Yaskawa INFORM job: A_ROOF_SIDE_0617_2_PAINT_38.JBI

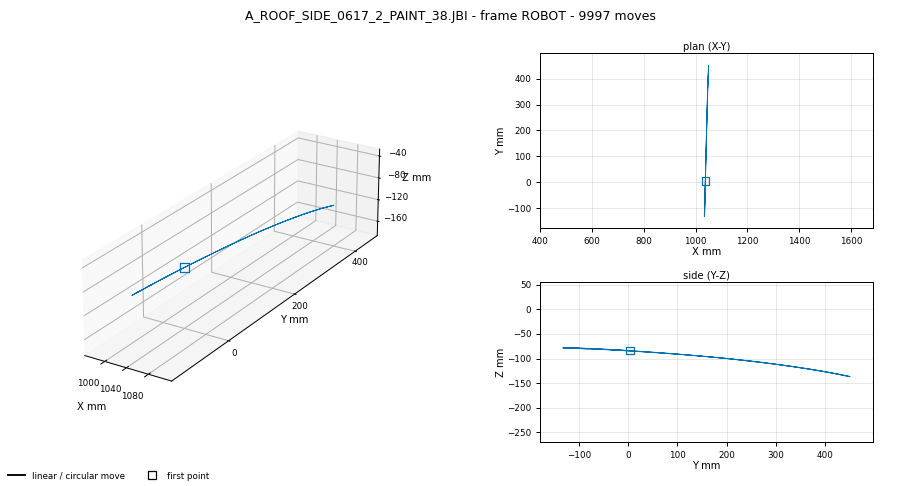
[picture p0: tool path of A_ROOF_SIDE_0617_2_PAINT_38.JBI in frame ROBOT, 9997 of 9997 moves have a stored position in this frame; points joined in program order, loops and branches not executed]
/JOB
//NAME A_ROOF_SIDE_0617_2_PAINT38
//POS
///NPOS 9997,0,0,0,0,0
///TOOL 1
///USER 0
///POSTYPE ROBOT
///RECTAN
///RCONF 1,0,0,0,0,0,0,0,0,0,0,0,0,0,0,0,0,0,0,0,0,0,0,0
C00000=1038.602,4.490,-83.697,169.159,38.320,157.198
C00001=1038.595,4.241,-83.682,169.157,38.319,157.198
C00002=1038.590,3.992,-83.668,169.155,38.320,157.198
C00003=1038.583,3.742,-83.653,169.153,38.319,157.198
C00004=1038.577,3.493,-83.638,169.151,38.318,157.198
C00005=1038.570,3.243,-83.622,169.149,38.318,157.198
C00006=1038.564,2.994,-83.607,169.147,38.318,157.198
C00007=1038.557,2.744,-83.592,169.145,38.317,157.197
C00008=1038.552,2.495,-83.578,169.142,38.317,157.197
C00009=1038.545,2.246,-83.563,169.140,38.317,157.197
C00010=1038.539,1.996,-83.548,169.138,38.316,157.197
C00011=1038.532,1.746,-83.533,169.136,38.316,157.197
C00012=1038.526,1.497,-83.518,169.134,38.315,157.197
C00013=1038.519,1.248,-83.502,169.132,38.315,157.197
C00014=1038.514,0.999,-83.487,169.130,38.315,157.197
C00015=1038.507,0.749,-83.473,169.128,38.314,157.197
C00016=1038.501,0.499,-83.458,169.125,38.314,157.196
C00017=1038.495,0.249,-83.442,169.123,38.314,157.196
C00018=1038.489,-0.000,-83.427,169.121,38.313,157.196
C00019=1038.483,-0.249,-83.413,169.119,38.313,157.196
C00020=1038.477,-0.499,-83.398,169.116,38.313,157.196
C00021=1038.470,-0.749,-83.383,169.114,38.312,157.196
C00022=1038.464,-0.998,-83.368,169.112,38.312,157.196
C00023=1038.458,-1.247,-83.353,169.110,38.311,157.196
C00024=1038.452,-1.497,-83.338,169.108,38.311,157.196
C00025=1038.445,-1.747,-83.323,169.106,38.311,157.196
C00026=1038.439,-1.996,-83.308,169.104,38.310,157.195
C00027=1038.433,-2.245,-83.294,169.102,38.310,157.195
C00028=1038.427,-2.495,-83.279,169.100,38.310,157.195
C00029=1038.420,-2.744,-83.264,169.098,38.309,157.195
C00030=1038.414,-2.994,-83.249,169.096,38.309,157.195
C00031=1038.407,-3.278,-83.233,169.092,38.308,157.195
C00032=1038.400,-3.560,-83.215,169.090,38.308,157.195
C00033=1038.393,-3.844,-83.198,169.087,38.308,157.195
C00034=1038.385,-4.127,-83.183,169.085,38.307,157.194
C00035=1038.379,-4.377,-83.168,169.083,38.307,157.194
C00036=1038.373,-4.627,-83.153,169.081,38.307,157.194
C00037=1038.366,-4.876,-83.138,169.079,38.307,157.194
C00038=1038.360,-5.125,-83.124,169.076,38.306,157.194
C00039=1038.354,-5.375,-83.110,169.074,38.306,157.194
C00040=1038.347,-5.625,-83.095,169.072,38.306,157.194
C00041=1038.340,-5.874,-83.080,169.070,38.306,157.194
C00042=1038.334,-6.123,-83.066,169.068,38.305,157.194
C00043=1038.328,-6.373,-83.051,169.066,38.306,157.194
C00044=1038.321,-6.623,-83.037,169.064,38.305,157.194
C00045=1038.315,-6.873,-83.022,169.061,38.304,157.193
C00046=1038.309,-7.122,-83.008,169.058,38.305,157.193
C00047=1038.303,-7.371,-82.993,169.056,38.304,157.193
C00048=1038.296,-7.621,-82.979,169.054,38.304,157.193
C00049=1038.290,-7.870,-82.965,169.052,38.304,157.193
C00050=1038.284,-8.120,-82.950,169.050,38.304,157.193
C00051=1038.277,-8.369,-82.935,169.048,38.303,157.193
C00052=1038.271,-8.619,-82.921,169.046,38.303,157.193
C00053=1038.265,-8.868,-82.906,169.043,38.303,157.193
C00054=1038.258,-9.118,-82.892,169.041,38.303,157.193
C00055=1038.252,-9.367,-82.877,169.039,38.302,157.193
C00056=1038.246,-9.617,-82.863,169.037,38.302,157.192
C00057=1038.239,-9.866,-82.849,169.035,38.302,157.192
C00058=1038.233,-10.115,-82.834,169.033,38.301,157.192
C00059=1038.227,-10.365,-82.820,169.030,38.301,157.192
C00060=1038.220,-10.615,-82.806,169.027,38.301,157.192
C00061=1038.214,-10.864,-82.791,169.025,38.301,157.192
C00062=1038.208,-11.114,-82.777,169.023,38.300,157.192
C00063=1038.201,-11.363,-82.763,169.021,38.300,157.192
C00064=1038.195,-11.613,-82.749,169.019,38.300,157.192
C00065=1038.189,-11.863,-82.734,169.017,38.299,157.192
C00066=1038.182,-12.111,-82.720,169.015,38.299,157.192
C00067=1038.176,-12.362,-82.706,169.012,38.299,157.191
C00068=1038.170,-12.611,-82.691,169.010,38.299,157.191
C00069=1038.163,-12.860,-82.677,169.008,38.298,157.191
C00070=1038.157,-13.110,-82.662,169.006,38.299,157.191
C00071=1038.151,-13.359,-82.648,169.004,38.298,157.191
C00072=1038.145,-13.609,-82.634,169.002,38.298,157.191
C00073=1038.139,-13.858,-82.620,168.998,38.298,157.191
C00074=1038.132,-14.108,-82.606,168.996,38.298,157.191
C00075=1038.126,-14.358,-82.591,168.994,38.297,157.191
C00076=1038.120,-14.607,-82.577,168.992,38.297,157.191
C00077=1038.113,-14.857,-82.563,168.990,38.297,157.191
C00078=1038.107,-15.105,-82.548,168.988,38.296,157.190
C00079=1038.101,-15.356,-82.534,168.985,38.296,157.190
C00080=1038.095,-15.605,-82.521,168.983,38.296,157.190
C00081=1038.088,-15.854,-82.506,168.981,38.296,157.190
C00082=1038.082,-16.105,-82.492,168.979,38.296,157.190
C00083=1038.075,-16.353,-82.478,168.977,38.295,157.190
C00084=1038.069,-16.604,-82.464,168.974,38.295,157.190
C00085=1038.063,-16.852,-82.450,168.972,38.295,157.190
C00086=1038.056,-17.102,-82.436,168.970,38.295,157.190
C00087=1038.050,-17.352,-82.422,168.968,38.294,157.190
C00088=1038.043,-17.601,-82.408,168.966,38.295,157.190
C00089=1038.037,-17.851,-82.394,168.963,38.295,157.190
C00090=1038.031,-18.100,-82.380,168.960,38.294,157.190
C00091=1038.024,-18.350,-82.366,168.958,38.294,157.190
C00092=1038.018,-18.600,-82.352,168.956,38.294,157.189
C00093=1038.011,-18.849,-82.338,168.954,38.294,157.189
C00094=1038.005,-19.098,-82.325,168.951,38.294,157.189
C00095=1037.998,-19.380,-82.308,168.949,38.293,157.189
C00096=1037.992,-19.662,-82.293,168.946,38.293,157.189
C00097=1037.984,-19.944,-82.277,168.944,38.293,157.189
C00098=1037.977,-20.226,-82.262,168.941,38.293,157.189
C00099=1037.970,-20.475,-82.248,168.939,38.292,157.189
C00100=1037.964,-20.725,-82.234,168.937,38.293,157.189
C00101=1037.958,-20.975,-82.220,168.935,38.293,157.189
C00102=1037.951,-21.224,-82.206,168.932,38.292,157.189
C00103=1037.945,-21.473,-82.192,168.930,38.292,157.189
C00104=1037.939,-21.723,-82.178,168.928,38.292,157.188
C00105=1037.932,-21.973,-82.165,168.926,38.292,157.188
C00106=1037.926,-22.223,-82.151,168.923,38.291,157.188
C00107=1037.920,-22.472,-82.137,168.920,38.291,157.188
C00108=1037.914,-22.721,-82.123,168.918,38.291,157.188
C00109=1037.908,-22.971,-82.109,168.916,38.291,157.188
C00110=1037.901,-23.220,-82.096,168.914,38.291,157.188
C00111=1037.894,-23.470,-82.082,168.911,38.290,157.188
C00112=1037.889,-23.719,-82.068,168.909,38.291,157.188
C00113=1037.882,-23.969,-82.054,168.907,38.291,157.188
C00114=1037.876,-24.219,-82.041,168.905,38.290,157.188
C00115=1037.870,-24.468,-82.027,168.903,38.290,157.188
C00116=1037.863,-24.717,-82.013,168.900,38.290,157.188
C00117=1037.857,-24.967,-81.999,168.898,38.290,157.188
C00118=1037.851,-25.217,-81.985,168.896,38.290,157.188
C00119=1037.845,-25.466,-81.972,168.894,38.289,157.187
C00120=1037.838,-25.716,-81.959,168.891,38.289,157.187
C00121=1037.832,-25.966,-81.944,168.889,38.289,157.187
C00122=1037.826,-26.215,-81.931,168.887,38.289,157.187
C00123=1037.820,-26.464,-81.918,168.885,38.288,157.187
C00124=1037.813,-26.714,-81.903,168.881,38.289,157.187
C00125=1037.807,-26.963,-81.890,168.879,38.289,157.187
C00126=1037.800,-27.213,-81.876,168.877,38.288,157.187
C00127=1037.794,-27.462,-81.863,168.875,38.288,157.187
C00128=1037.789,-27.712,-81.849,168.872,38.288,157.187
C00129=1037.782,-27.962,-81.835,168.870,38.288,157.187
C00130=1037.776,-28.211,-81.822,168.868,38.288,157.187
C00131=1037.769,-28.461,-81.809,168.865,38.288,157.187
C00132=1037.763,-28.711,-81.795,168.863,38.288,157.187
C00133=1037.756,-28.960,-81.782,168.861,38.288,157.187
C00134=1037.750,-29.210,-81.768,168.859,38.288,157.186
C00135=1037.743,-29.459,-81.755,168.856,38.288,157.186
C00136=1037.737,-29.708,-81.742,168.854,38.288,157.186
C00137=1037.731,-29.959,-81.729,168.852,38.287,157.186
C00138=1037.725,-30.208,-81.715,168.849,38.287,157.186
C00139=1037.718,-30.457,-81.702,168.847,38.288,157.186
C00140=1037.712,-30.708,-81.688,168.845,38.288,157.186
C00141=1037.706,-30.957,-81.675,168.843,38.287,157.186
C00142=1037.700,-31.206,-81.661,168.840,38.287,157.186
C00143=1037.693,-31.456,-81.648,168.838,38.287,157.186
C00144=1037.687,-31.705,-81.634,168.836,38.287,157.186
C00145=1037.681,-31.955,-81.621,168.833,38.287,157.186
C00146=1037.674,-32.204,-81.608,168.831,38.287,157.186
C00147=1037.668,-32.455,-81.595,168.829,38.287,157.186
C00148=1037.662,-32.704,-81.582,168.826,38.287,157.186
C00149=1037.655,-32.953,-81.568,168.823,38.287,157.185
C00150=1037.649,-33.203,-81.555,168.821,38.287,157.185
C00151=1037.642,-33.452,-81.542,168.819,38.287,157.185
C00152=1037.636,-33.702,-81.528,168.816,38.287,157.185
C00153=1037.630,-33.951,-81.515,168.814,38.286,157.185
C00154=1037.623,-34.201,-81.502,168.812,38.287,157.185
C00155=1037.617,-34.451,-81.489,168.809,38.287,157.185
C00156=1037.611,-34.700,-81.476,168.807,38.287,157.185
C00157=1037.605,-34.949,-81.462,168.805,38.286,157.185
C00158=1037.598,-35.200,-81.449,168.802,38.286,157.185
C00159=1037.592,-35.480,-81.434,168.800,38.286,157.185
C00160=1037.585,-35.762,-81.420,168.797,38.287,157.185
C00161=1037.578,-36.043,-81.404,168.795,38.286,157.185
C00162=1037.571,-36.323,-81.390,168.792,38.286,157.185
C00163=1037.564,-36.573,-81.376,168.790,38.286,157.185
C00164=1037.558,-36.823,-81.363,168.787,38.286,157.185
C00165=1037.552,-37.073,-81.350,168.785,38.286,157.185
C00166=1037.546,-37.322,-81.337,168.783,38.286,157.185
C00167=1037.540,-37.571,-81.324,168.780,38.286,157.184
C00168=1037.533,-37.822,-81.311,168.778,38.286,157.184
C00169=1037.527,-38.071,-81.298,168.776,38.286,157.184
C00170=1037.521,-38.320,-81.284,168.773,38.286,157.184
C00171=1037.515,-38.570,-81.272,168.771,38.286,157.184
C00172=1037.508,-38.819,-81.258,168.769,38.286,157.184
C00173=1037.502,-39.069,-81.245,168.766,38.286,157.184
C00174=1037.496,-39.319,-81.232,168.763,38.286,157.184
C00175=1037.490,-39.568,-81.219,168.761,38.286,157.184
C00176=1037.483,-39.818,-81.207,168.758,38.286,157.184
C00177=1037.477,-40.067,-81.194,168.756,38.286,157.184
C00178=1037.470,-40.317,-81.180,168.754,38.286,157.184
C00179=1037.465,-40.566,-81.168,168.751,38.286,157.184
C00180=1037.458,-40.816,-81.154,168.749,38.286,157.184
C00181=1037.451,-41.066,-81.142,168.746,38.286,157.184
C00182=1037.445,-41.315,-81.129,168.744,38.286,157.184
C00183=1037.439,-41.565,-81.117,168.742,38.286,157.184
C00184=1037.433,-41.814,-81.103,168.739,38.287,157.184
C00185=1037.426,-42.064,-81.091,168.737,38.286,157.184
C00186=1037.420,-42.313,-81.078,168.735,38.286,157.184
C00187=1037.413,-42.564,-81.065,168.732,38.286,157.184
C00188=1037.407,-42.813,-81.052,168.730,38.286,157.184
C00189=1037.401,-43.063,-81.040,168.727,38.287,157.184
C00190=1037.394,-43.312,-81.027,168.725,38.287,157.184
C00191=1037.388,-43.562,-81.014,168.723,38.287,157.183
C00192=1037.382,-43.811,-81.001,168.720,38.287,157.183
C00193=1037.376,-44.061,-80.988,168.718,38.287,157.183
C00194=1037.370,-44.310,-80.976,168.716,38.287,157.183
C00195=1037.363,-44.560,-80.963,168.713,38.287,157.183
C00196=1037.358,-44.810,-80.950,168.711,38.287,157.183
C00197=1037.351,-45.059,-80.937,168.708,38.287,157.183
C00198=1037.345,-45.308,-80.925,168.706,38.287,157.183
C00199=1037.338,-45.559,-80.912,168.704,38.287,157.183
C00200=1037.332,-45.808,-80.899,168.701,38.287,157.183
C00201=1037.325,-46.058,-80.887,168.699,38.287,157.183
C00202=1037.319,-46.307,-80.874,168.696,38.287,157.183
C00203=1037.313,-46.557,-80.861,168.694,38.287,157.183
C00204=1037.307,-46.807,-80.849,168.692,38.288,157.183
C00205=1037.300,-47.056,-80.836,168.689,38.288,157.183
C00206=1037.294,-47.306,-80.823,168.687,38.288,157.183
C00207=1037.288,-47.556,-80.811,168.684,38.288,157.183
C00208=1037.282,-47.805,-80.798,168.682,38.288,157.183
C00209=1037.276,-48.054,-80.786,168.680,38.288,157.183
C00210=1037.270,-48.304,-80.773,168.677,38.288,157.183
C00211=1037.264,-48.554,-80.761,168.675,38.288,157.183
C00212=1037.257,-48.803,-80.748,168.673,38.288,157.183
C00213=1037.251,-49.053,-80.735,168.670,38.288,157.183
C00214=1037.245,-49.303,-80.723,168.668,38.288,157.183
C00215=1037.239,-49.552,-80.710,168.665,38.288,157.183
C00216=1037.232,-49.802,-80.698,168.663,38.288,157.183
C00217=1037.227,-50.051,-80.685,168.659,38.288,157.183
C00218=1037.221,-50.301,-80.673,168.657,38.288,157.182
C00219=1037.214,-50.550,-80.661,168.655,38.289,157.182
C00220=1037.208,-50.800,-80.648,168.652,38.289,157.182
C00221=1037.201,-51.049,-80.636,168.650,38.289,157.182
C00222=1037.196,-51.299,-80.623,168.648,38.290,157.182
C00223=1037.188,-51.581,-80.610,168.646,38.290,157.182
C00224=1037.180,-51.862,-80.596,168.642,38.290,157.182
C00225=1037.173,-52.144,-80.582,168.639,38.290,157.182
C00226=1037.166,-52.426,-80.567,168.636,38.290,157.182
C00227=1037.160,-52.675,-80.556,168.635,38.291,157.182
C00228=1037.153,-52.924,-80.544,168.632,38.291,157.182
C00229=1037.147,-53.174,-80.531,168.630,38.291,157.182
C00230=1037.141,-53.424,-80.519,168.626,38.291,157.182
C00231=1037.134,-53.673,-80.507,168.624,38.291,157.182
C00232=1037.128,-53.923,-80.495,168.621,38.291,157.182
C00233=1037.122,-54.173,-80.483,168.620,38.292,157.182
C00234=1037.115,-54.422,-80.471,168.617,38.292,157.182
C00235=1037.109,-54.672,-80.458,168.615,38.292,157.182
C00236=1037.102,-54.922,-80.446,168.612,38.293,157.182
C00237=1037.096,-55.172,-80.434,168.609,38.293,157.182
C00238=1037.090,-55.421,-80.422,168.607,38.293,157.182
C00239=1037.083,-55.671,-80.410,168.605,38.294,157.182
C00240=1037.077,-55.921,-80.397,168.602,38.294,157.182
C00241=1037.071,-56.170,-80.385,168.600,38.294,157.182
C00242=1037.065,-56.419,-80.374,168.597,38.294,157.182
C00243=1037.059,-56.669,-80.361,168.595,38.295,157.182
C00244=1037.052,-56.919,-80.349,168.592,38.295,157.182
C00245=1037.045,-57.168,-80.337,168.590,38.295,157.182
C00246=1037.039,-57.418,-80.325,168.588,38.295,157.182
C00247=1037.033,-57.668,-80.313,168.585,38.295,157.182
C00248=1037.026,-57.918,-80.302,168.583,38.296,157.182
C00249=1037.020,-58.167,-80.290,168.580,38.296,157.182
C00250=1037.014,-58.416,-80.277,168.578,38.296,157.182
C00251=1037.008,-58.666,-80.265,168.575,38.296,157.182
C00252=1037.001,-58.916,-80.254,168.573,38.296,157.182
C00253=1036.995,-59.166,-80.241,168.570,38.297,157.182
C00254=1036.989,-59.415,-80.229,168.568,38.297,157.182
C00255=1036.983,-59.664,-80.217,168.565,38.297,157.182
C00256=1036.977,-59.914,-80.206,168.563,38.297,157.182
C00257=1036.970,-60.164,-80.194,168.560,38.298,157.182
C00258=1036.964,-60.414,-80.182,168.558,38.298,157.182
C00259=1036.958,-60.663,-80.169,168.555,38.298,157.182
C00260=1036.952,-60.912,-80.157,168.553,38.299,157.182
C00261=1036.945,-61.163,-80.146,168.550,38.299,157.182
C00262=1036.939,-61.412,-80.134,168.548,38.299,157.182
C00263=1036.933,-61.662,-80.122,168.545,38.300,157.182
C00264=1036.926,-61.912,-80.110,168.543,38.300,157.182
C00265=1036.920,-62.160,-80.098,168.540,38.300,157.182
C00266=1036.915,-62.411,-80.086,168.538,38.300,157.182
C00267=1036.908,-62.661,-80.074,168.535,38.301,157.182
C00268=1036.901,-62.910,-80.062,168.533,38.301,157.182
C00269=1036.895,-63.159,-80.051,168.530,38.301,157.182
C00270=1036.890,-63.409,-80.039,168.527,38.301,157.182
C00271=1036.883,-63.659,-80.027,168.525,38.302,157.182
C00272=1036.877,-63.908,-80.015,168.522,38.302,157.182
C00273=1036.871,-64.158,-80.004,168.520,38.302,157.182
C00274=1036.865,-64.408,-79.992,168.517,38.302,157.182
C00275=1036.858,-64.658,-79.980,168.515,38.303,157.182
C00276=1036.852,-64.907,-79.969,168.512,38.303,157.182
C00277=1036.846,-65.157,-79.956,168.510,38.303,157.182
C00278=1036.840,-65.407,-79.944,168.507,38.303,157.182
C00279=1036.834,-65.656,-79.933,168.505,38.303,157.182
C00280=1036.827,-65.906,-79.921,168.502,38.304,157.182
C00281=1036.821,-66.155,-79.909,168.500,38.304,157.182
C00282=1036.816,-66.405,-79.898,168.497,38.304,157.182
C00283=1036.809,-66.655,-79.886,168.495,38.305,157.182
C00284=1036.802,-66.904,-79.874,168.492,38.305,157.182
C00285=1036.797,-67.154,-79.863,168.490,38.305,157.182
C00286=1036.791,-67.403,-79.851,168.487,38.306,157.182
C00287=1036.784,-67.686,-79.838,168.484,38.306,157.182
C00288=1036.777,-67.969,-79.825,168.481,38.307,157.182
C00289=1036.770,-68.252,-79.811,168.479,38.307,157.182
C00290=1036.763,-68.535,-79.798,168.476,38.307,157.182
C00291=1036.757,-68.784,-79.786,168.473,38.308,157.182
C00292=1036.751,-69.034,-79.775,168.471,38.308,157.182
C00293=1036.745,-69.284,-79.763,168.468,38.308,157.182
C00294=1036.739,-69.533,-79.752,168.466,38.308,157.182
C00295=1036.733,-69.783,-79.740,168.463,38.309,157.182
C00296=1036.726,-70.033,-79.729,168.461,38.309,157.182
C00297=1036.720,-70.282,-79.717,168.458,38.309,157.182
C00298=1036.715,-70.532,-79.705,168.455,38.309,157.182
C00299=1036.708,-70.781,-79.694,168.453,38.310,157.182
C00300=1036.702,-71.032,-79.683,168.450,38.310,157.182
C00301=1036.696,-71.280,-79.671,168.448,38.310,157.182
C00302=1036.690,-71.531,-79.659,168.445,38.311,157.182
C00303=1036.684,-71.780,-79.648,168.443,38.311,157.182
C00304=1036.678,-72.030,-79.636,168.440,38.311,157.182
C00305=1036.672,-72.279,-79.625,168.438,38.311,157.182
C00306=1036.666,-72.529,-79.613,168.435,38.312,157.182
C00307=1036.661,-72.779,-79.602,168.433,38.312,157.182
C00308=1036.654,-73.028,-79.590,168.430,38.312,157.182
C00309=1036.648,-73.278,-79.579,168.428,38.312,157.182
C00310=1036.642,-73.528,-79.568,168.425,38.313,157.182
C00311=1036.635,-73.778,-79.556,168.422,38.313,157.182
C00312=1036.630,-74.027,-79.545,168.420,38.313,157.182
C00313=1036.624,-74.278,-79.533,168.417,38.314,157.182
C00314=1036.617,-74.526,-79.522,168.415,38.314,157.182
C00315=1036.611,-74.776,-79.511,168.412,38.315,157.182
C00316=1036.605,-75.026,-79.500,168.410,38.315,157.182
C00317=1036.598,-75.275,-79.488,168.407,38.316,157.182
C00318=1036.593,-75.525,-79.477,168.404,38.316,157.182
C00319=1036.586,-75.775,-79.466,168.402,38.317,157.182
C00320=1036.581,-76.025,-79.455,168.399,38.317,157.182
C00321=1036.574,-76.274,-79.443,168.397,38.318,157.182
C00322=1036.568,-76.524,-79.432,168.394,38.318,157.182
C00323=1036.562,-76.774,-79.421,168.392,38.319,157.182
C00324=1036.556,-77.023,-79.410,168.390,38.319,157.182
C00325=1036.550,-77.274,-79.399,168.387,38.320,157.182
C00326=1036.544,-77.522,-79.387,168.385,38.320,157.182
C00327=1036.537,-77.773,-79.376,168.382,38.320,157.183
C00328=1036.531,-78.022,-79.366,168.379,38.321,157.182
C00329=1036.525,-78.271,-79.355,168.377,38.321,157.183
C00330=1036.519,-78.521,-79.344,168.374,38.321,157.183
C00331=1036.513,-78.771,-79.333,168.372,38.322,157.183
C00332=1036.507,-79.021,-79.321,168.369,38.322,157.183
C00333=1036.501,-79.270,-79.310,168.366,38.323,157.183
C00334=1036.494,-79.520,-79.299,168.364,38.323,157.183
C00335=1036.489,-79.770,-79.288,168.361,38.324,157.183
C00336=1036.483,-80.019,-79.277,168.359,38.324,157.183
C00337=1036.476,-80.269,-79.266,168.356,38.325,157.183
C00338=1036.470,-80.519,-79.256,168.353,38.325,157.183
C00339=1036.464,-80.769,-79.244,168.351,38.326,157.183
C00340=1036.457,-81.018,-79.234,168.348,38.327,157.183
C00341=1036.451,-81.268,-79.223,168.345,38.327,157.183
C00342=1036.445,-81.518,-79.212,168.343,38.328,157.183
C00343=1036.438,-81.767,-79.201,168.340,38.328,157.183
C00344=1036.432,-82.017,-79.190,168.337,38.329,157.183
C00345=1036.427,-82.266,-79.179,168.335,38.329,157.183
C00346=1036.420,-82.516,-79.169,168.333,38.330,157.183
C00347=1036.414,-82.766,-79.158,168.330,38.331,157.183
C00348=1036.408,-83.016,-79.147,168.328,38.331,157.183
C00349=1036.401,-83.265,-79.136,168.325,38.332,157.183
C00350=1036.395,-83.515,-79.126,168.322,38.333,157.183
C00351=1036.388,-83.800,-79.113,168.319,38.333,157.183
C00352=1036.381,-84.085,-79.101,168.316,38.334,157.183
C00353=1036.374,-84.370,-79.089,168.313,38.334,157.184
C00354=1036.367,-84.655,-79.077,168.310,38.335,157.184
C00355=1036.361,-84.905,-79.066,168.308,38.336,157.184
C00356=1036.354,-85.154,-79.056,168.305,38.336,157.184
C00357=1036.349,-85.404,-79.045,168.302,38.337,157.184
C00358=1036.342,-85.654,-79.033,168.300,38.338,157.184
C00359=1036.336,-85.903,-79.023,168.297,38.338,157.184
C00360=1036.330,-86.152,-79.012,168.294,38.339,157.184
C00361=1036.323,-86.402,-79.002,168.292,38.339,157.184
C00362=1036.318,-86.652,-78.991,168.289,38.340,157.184
C00363=1036.312,-86.902,-78.981,168.286,38.340,157.184
C00364=1036.305,-87.152,-78.970,168.285,38.341,157.184
C00365=1036.299,-87.401,-78.959,168.282,38.342,157.184
C00366=1036.293,-87.651,-78.948,168.279,38.343,157.184
C00367=1036.287,-87.901,-78.939,168.277,38.343,157.184
C00368=1036.281,-88.151,-78.927,168.274,38.343,157.184
C00369=1036.274,-88.400,-78.917,168.271,38.344,157.184
C00370=1036.269,-88.649,-78.906,168.268,38.345,157.184
C00371=1036.263,-88.900,-78.896,168.266,38.345,157.184
C00372=1036.256,-89.149,-78.885,168.263,38.346,157.185
C00373=1036.250,-89.399,-78.874,168.260,38.347,157.185
C00374=1036.244,-89.648,-78.864,168.258,38.348,157.185
C00375=1036.238,-89.899,-78.854,168.255,38.348,157.185
C00376=1036.232,-90.148,-78.843,168.252,38.349,157.185
C00377=1036.226,-90.398,-78.833,168.250,38.349,157.185
C00378=1036.220,-90.648,-78.822,168.247,38.350,157.185
C00379=1036.214,-90.897,-78.812,168.244,38.350,157.185
C00380=1036.207,-91.147,-78.801,168.242,38.351,157.185
C00381=1036.201,-91.396,-78.791,168.240,38.352,157.185
C00382=1036.195,-91.646,-78.780,168.237,38.353,157.185
C00383=1036.190,-91.896,-78.770,168.235,38.353,157.185
C00384=1036.184,-92.146,-78.760,168.232,38.353,157.185
C00385=1036.178,-92.395,-78.749,168.229,38.354,157.185
///RCONF 1,0,0,0,1,0,0,0,0,0,0,0,0,0,0,0,0,0,0,0,0,0,0,0
C00386=1036.171,-92.645,-78.738,168.227,38.355,157.185
C00387=1036.165,-92.895,-78.728,168.224,38.355,157.185
C00388=1036.160,-93.145,-78.717,168.221,38.356,157.185
C00389=1036.153,-93.394,-78.707,168.219,38.357,157.185
C00390=1036.148,-93.644,-78.697,168.216,38.358,157.186
C00391=1036.141,-93.893,-78.687,168.213,38.358,157.186
C00392=1036.135,-94.144,-78.676,168.211,38.358,157.186
C00393=1036.129,-94.393,-78.666,168.208,38.359,157.186
C00394=1036.123,-94.643,-78.656,168.205,38.360,157.186
C00395=1036.117,-94.892,-78.645,168.202,38.361,157.186
C00396=1036.111,-95.142,-78.635,168.200,38.361,157.186
C00397=1036.106,-95.392,-78.624,168.197,38.362,157.186
C00398=1036.099,-95.641,-78.614,168.195,38.363,157.186
C00399=1036.094,-95.891,-78.604,168.193,38.363,157.186
C00400=1036.087,-96.140,-78.594,168.190,38.364,157.186
C00401=1036.082,-96.390,-78.583,168.187,38.364,157.186
C00402=1036.075,-96.640,-78.573,168.185,38.365,157.186
C00403=1036.069,-96.890,-78.563,168.182,38.366,157.186
C00404=1036.063,-97.140,-78.552,168.179,38.367,157.186
C00405=1036.057,-97.390,-78.542,168.177,38.367,157.186
C00406=1036.051,-97.640,-78.533,168.174,38.368,157.187
C00407=1036.045,-97.889,-78.522,168.171,38.369,157.187
C00408=1036.039,-98.139,-78.512,168.168,38.370,157.187
C00409=1036.033,-98.388,-78.502,168.166,38.371,157.187
C00410=1036.027,-98.638,-78.492,168.163,38.371,157.187
C00411=1036.021,-98.888,-78.482,168.161,38.372,157.187
C00412=1036.015,-99.137,-78.472,168.158,38.373,157.187
C00413=1036.008,-99.387,-78.462,168.156,38.374,157.187
C00414=1036.002,-99.638,-78.452,168.153,38.375,157.187
C00415=1035.993,-100.042,-78.436,168.148,38.376,157.187
C00416=1035.983,-100.445,-78.419,168.144,38.377,157.187
C00417=1035.972,-100.849,-78.403,168.140,38.378,157.187
C00418=1035.963,-101.253,-78.387,168.135,38.379,157.188
C00419=1035.957,-101.503,-78.377,168.132,38.380,157.188
C00420=1035.951,-101.753,-78.368,168.130,38.381,157.188
C00421=1035.945,-102.002,-78.358,168.128,38.382,157.188
C00422=1035.938,-102.252,-78.348,168.125,38.383,157.188
C00423=1035.933,-102.502,-78.337,168.122,38.383,157.188
C00424=1035.927,-102.752,-78.328,168.120,38.384,157.188
C00425=1035.921,-103.001,-78.318,168.117,38.385,157.188
C00426=1035.914,-103.251,-78.308,168.114,38.386,157.188
C00427=1035.909,-103.501,-78.298,168.111,38.387,157.188
C00428=1035.903,-103.750,-78.288,168.109,38.387,157.188
C00429=1035.896,-104.000,-78.279,168.106,38.388,157.189
C00430=1035.890,-104.250,-78.269,168.103,38.389,157.189
C00431=1035.885,-104.500,-78.259,168.101,38.391,157.189
C00432=1035.878,-104.749,-78.249,168.099,38.391,157.189
C00433=1035.872,-104.999,-78.239,168.096,38.392,157.189
C00434=1035.867,-105.248,-78.230,168.093,38.393,157.189
C00435=1035.861,-105.498,-78.220,168.090,38.394,157.189
C00436=1035.855,-105.748,-78.210,168.088,38.394,157.189
C00437=1035.849,-105.998,-78.201,168.085,38.395,157.189
C00438=1035.843,-106.248,-78.191,168.082,38.396,157.189
C00439=1035.833,-106.631,-78.175,168.078,38.398,157.190
C00440=1035.824,-107.013,-78.161,168.074,38.399,157.190
C00441=1035.815,-107.396,-78.146,168.070,38.400,157.190
C00442=1035.806,-107.778,-78.132,168.066,38.402,157.190
C00443=1035.799,-108.027,-78.122,168.063,38.402,157.190
C00444=1035.794,-108.278,-78.112,168.061,38.403,157.190
C00445=1035.788,-108.527,-78.102,168.058,38.405,157.190
C00446=1035.782,-108.777,-78.093,168.055,38.405,157.190
C00447=1035.775,-109.027,-78.083,168.052,38.406,157.190
C00448=1035.769,-109.277,-78.074,168.049,38.407,157.191
C00449=1035.763,-109.527,-78.064,168.047,38.408,157.191
C00450=1035.757,-109.776,-78.055,168.045,38.409,157.191
C00451=1035.751,-110.025,-78.045,168.042,38.410,157.191
C00452=1035.745,-110.276,-78.036,168.039,38.411,157.191
C00453=1035.739,-110.526,-78.027,168.036,38.412,157.191
C00454=1035.733,-110.775,-78.017,168.034,38.413,157.191
C00455=1035.727,-111.025,-78.008,168.031,38.414,157.191
C00456=1035.721,-111.275,-77.998,168.028,38.415,157.191
C00457=1035.715,-111.524,-77.989,168.025,38.416,157.191
C00458=1035.709,-111.774,-77.979,168.022,38.417,157.192
C00459=1035.703,-112.024,-77.970,168.021,38.418,157.192
C00460=1035.697,-112.274,-77.960,168.018,38.419,157.192
C00461=1035.691,-112.523,-77.951,168.015,38.419,157.192
C00462=1035.685,-112.773,-77.942,168.012,38.421,157.192
C00463=1035.679,-113.023,-77.933,168.009,38.422,157.192
C00464=1035.673,-113.273,-77.923,168.007,38.423,157.192
C00465=1035.667,-113.522,-77.914,168.004,38.423,157.192
C00466=1035.661,-113.772,-77.904,168.001,38.425,157.193
C00467=1035.655,-114.021,-77.895,167.998,38.426,157.193
C00468=1035.649,-114.272,-77.886,167.996,38.426,157.193
C00469=1035.643,-114.522,-77.876,167.994,38.427,157.193
C00470=1035.637,-114.771,-77.867,167.991,38.429,157.193
C00471=1035.631,-115.020,-77.858,167.988,38.430,157.193
C00472=1035.625,-115.271,-77.849,167.985,38.430,157.193
C00473=1035.619,-115.521,-77.839,167.982,38.432,157.193
C00474=1035.613,-115.770,-77.830,167.980,38.433,157.193
C00475=1035.606,-116.056,-77.820,167.976,38.434,157.194
C00476=1035.599,-116.343,-77.809,167.973,38.435,157.194
C00477=1035.593,-116.629,-77.798,167.971,38.436,157.194
C00478=1035.586,-116.916,-77.788,167.968,38.437,157.194
C00479=1035.579,-117.166,-77.779,167.965,38.439,157.194
C00480=1035.573,-117.416,-77.769,167.962,38.440,157.194
C00481=1035.568,-117.666,-77.761,167.959,38.440,157.194
C00482=1035.562,-117.915,-77.751,167.956,38.442,157.194
C00483=1035.556,-118.165,-77.742,167.954,38.443,157.194
C00484=1035.550,-118.415,-77.733,167.952,38.444,157.195
C00485=1035.543,-118.664,-77.724,167.949,38.445,157.195
C00486=1035.537,-118.914,-77.715,167.946,38.446,157.195
C00487=1035.532,-119.164,-77.706,167.943,38.447,157.195
C00488=1035.526,-119.414,-77.697,167.940,38.448,157.195
C00489=1035.520,-119.664,-77.688,167.938,38.449,157.195
C00490=1035.514,-119.913,-77.679,167.935,38.450,157.195
C00491=1035.508,-120.163,-77.670,167.932,38.452,157.196
C00492=1035.502,-120.413,-77.661,167.930,38.453,157.196
C00493=1035.496,-120.662,-77.651,167.927,38.454,157.196
C00494=1035.490,-120.913,-77.643,167.924,38.455,157.196
C00495=1035.484,-121.162,-77.633,167.922,38.456,157.196
C00496=1035.478,-121.412,-77.625,167.919,38.457,157.196
C00497=1035.472,-121.662,-77.616,167.916,38.458,157.196
C00498=1035.467,-121.911,-77.607,167.913,38.459,157.196
C00499=1035.460,-122.161,-77.598,167.910,38.460,157.197
C00500=1035.455,-122.412,-77.589,167.908,38.462,157.197
C00501=1035.448,-122.660,-77.580,167.906,38.463,157.197
C00502=1035.442,-122.911,-77.571,167.903,38.464,157.197
C00503=1035.437,-123.160,-77.562,167.900,38.465,157.197
C00504=1035.431,-123.410,-77.553,167.897,38.466,157.197
C00505=1035.424,-123.660,-77.544,167.894,38.467,157.197
C00506=1035.419,-123.909,-77.536,167.891,38.469,157.198
C00507=1035.413,-124.160,-77.527,167.890,38.469,157.198
C00508=1035.407,-124.409,-77.518,167.887,38.471,157.198
C00509=1035.401,-124.659,-77.509,167.884,38.472,157.198
C00510=1035.395,-124.908,-77.500,167.881,38.473,157.198
C00511=1035.389,-125.159,-77.491,167.878,38.475,157.198
C00512=1035.383,-125.409,-77.483,167.875,38.475,157.198
C00513=1035.377,-125.658,-77.474,167.872,38.477,157.199
C00514=1035.371,-125.908,-77.465,167.870,38.478,157.199
C00515=1035.365,-126.158,-77.457,167.868,38.479,157.199
C00516=1035.359,-126.407,-77.448,167.865,38.481,157.199
C00517=1035.353,-126.657,-77.440,167.862,38.482,157.199
C00518=1035.347,-126.907,-77.431,167.859,38.483,157.199
C00519=1035.342,-127.156,-77.422,167.856,38.484,157.199
C00520=1035.335,-127.406,-77.413,167.853,38.485,157.199
C00521=1035.330,-127.656,-77.405,167.851,38.487,157.200
C00522=1035.324,-127.906,-77.395,167.849,38.488,157.200
C00523=1035.318,-128.156,-77.387,167.846,38.488,157.200
C00524=1035.314,-128.405,-77.376,167.843,38.489,157.200
C00525=1035.311,-128.654,-77.366,167.841,38.489,157.200
C00526=1035.307,-128.904,-77.355,167.839,38.488,157.200
C00527=1035.305,-129.155,-77.344,167.836,38.487,157.199
C00528=1035.303,-129.404,-77.331,167.834,38.485,157.199
C00529=1035.303,-129.654,-77.319,167.832,38.483,157.199
C00530=1035.303,-129.904,-77.305,167.830,38.480,157.198
C00531=1035.303,-130.155,-77.291,167.829,38.478,157.198
C00532=1035.304,-130.404,-77.277,167.827,38.474,157.197
C00533=1035.307,-130.654,-77.261,167.826,38.471,157.196
C00534=1035.309,-130.903,-77.245,167.824,38.466,157.196
C00535=1035.313,-131.154,-77.230,167.822,38.461,157.195
C00536=1035.317,-131.404,-77.212,167.821,38.456,157.194
C00537=1035.322,-131.655,-77.194,167.820,38.451,157.193
C00538=1035.327,-131.904,-77.176,167.819,38.444,157.192
C00539=1034.993,-131.929,-77.456,167.770,38.661,157.227
C00540=1034.988,-131.679,-77.475,167.771,38.667,157.228
C00541=1034.983,-131.429,-77.492,167.772,38.673,157.229
C00542=1034.979,-131.179,-77.509,167.774,38.678,157.230
C00543=1034.975,-130.928,-77.525,167.775,38.683,157.231
C00544=1034.973,-130.678,-77.541,167.777,38.687,157.232
C00545=1034.971,-130.429,-77.557,167.778,38.691,157.232
C00546=1034.969,-130.179,-77.571,167.780,38.695,157.233
C00547=1034.968,-129.929,-77.585,167.782,38.697,157.233
C00548=1034.969,-129.679,-77.599,167.784,38.700,157.234
C00549=1034.970,-129.429,-77.611,167.786,38.702,157.234
C00550=1034.971,-129.180,-77.623,167.788,38.704,157.235
C00551=1034.973,-128.929,-77.636,167.790,38.705,157.235
C00552=1034.977,-128.679,-77.647,167.793,38.706,157.235
C00553=1034.980,-128.430,-77.657,167.795,38.705,157.235
C00554=1034.984,-128.180,-77.667,167.797,38.705,157.235
C00555=1034.989,-127.930,-77.676,167.800,38.704,157.235
C00556=1034.996,-127.681,-77.685,167.803,38.704,157.235
C00557=1035.001,-127.431,-77.694,167.806,38.702,157.235
C00558=1035.008,-127.181,-77.703,167.808,38.701,157.235
C00559=1035.013,-126.932,-77.711,167.811,38.700,157.235
C00560=1035.019,-126.681,-77.720,167.814,38.698,157.234
C00561=1035.025,-126.433,-77.729,167.816,38.697,157.234
C00562=1035.031,-126.182,-77.737,167.819,38.696,157.234
C00563=1035.036,-125.932,-77.746,167.822,38.694,157.234
C00564=1035.043,-125.682,-77.754,167.824,38.693,157.234
C00565=1035.048,-125.433,-77.763,167.827,38.692,157.234
C00566=1035.054,-125.183,-77.772,167.830,38.691,157.233
C00567=1035.061,-124.934,-77.781,167.833,38.690,157.233
C00568=1035.066,-124.684,-77.790,167.836,38.688,157.233
C00569=1035.073,-124.434,-77.797,167.838,38.687,157.233
C00570=1035.079,-124.184,-77.807,167.841,38.686,157.233
C00571=1035.085,-123.934,-77.816,167.843,38.684,157.233
C00572=1035.090,-123.684,-77.824,167.846,38.684,157.233
C00573=1035.097,-123.435,-77.833,167.849,38.682,157.232
C00574=1035.102,-123.185,-77.842,167.852,38.681,157.232
C00575=1035.108,-122.935,-77.851,167.855,38.680,157.232
C00576=1035.113,-122.686,-77.860,167.857,38.679,157.232
C00577=1035.120,-122.436,-77.869,167.860,38.677,157.232
C00578=1035.126,-122.186,-77.878,167.862,38.677,157.232
C00579=1035.132,-121.937,-77.887,167.865,38.675,157.232
C00580=1035.138,-121.686,-77.896,167.868,38.674,157.232
C00581=1035.143,-121.437,-77.905,167.871,38.673,157.231
C00582=1035.150,-121.187,-77.913,167.874,38.671,157.231
C00583=1035.156,-120.937,-77.923,167.877,38.670,157.231
C00584=1035.161,-120.687,-77.931,167.879,38.669,157.231
C00585=1035.167,-120.438,-77.941,167.881,38.668,157.231
C00586=1035.173,-120.187,-77.950,167.884,38.667,157.231
C00587=1035.180,-119.938,-77.958,167.887,38.666,157.231
C00588=1035.185,-119.688,-77.967,167.890,38.665,157.231
C00589=1035.192,-119.438,-77.977,167.893,38.664,157.230
C00590=1035.197,-119.189,-77.986,167.895,38.663,157.230
C00591=1035.203,-118.939,-77.995,167.898,38.661,157.230
C00592=1035.209,-118.689,-78.004,167.901,38.660,157.230
C00593=1035.215,-118.439,-78.012,167.903,38.659,157.230
C00594=1035.221,-118.190,-78.022,167.906,38.658,157.230
C00595=1035.228,-117.940,-78.031,167.909,38.657,157.230
C00596=1035.233,-117.690,-78.040,167.912,38.656,157.230
C00597=1035.239,-117.440,-78.049,167.914,38.654,157.229
C00598=1035.245,-117.191,-78.059,167.917,38.653,157.229
C00599=1035.250,-116.941,-78.067,167.920,38.653,157.229
C00600=1035.258,-116.655,-78.078,167.922,38.651,157.229
C00601=1035.265,-116.368,-78.089,167.926,38.650,157.229
C00602=1035.271,-116.081,-78.100,167.929,38.649,157.229
C00603=1035.279,-115.795,-78.110,167.932,38.647,157.229
C00604=1035.285,-115.545,-78.119,167.935,38.646,157.229
C00605=1035.290,-115.296,-78.128,167.938,38.645,157.228
C00606=1035.296,-115.046,-78.137,167.941,38.644,157.228
C00607=1035.303,-114.796,-78.147,167.942,38.643,157.228
C00608=1035.308,-114.546,-78.156,167.945,38.642,157.228
C00609=1035.314,-114.296,-78.165,167.948,38.641,157.228
C00610=1035.320,-114.047,-78.175,167.951,38.640,157.228
C00611=1035.326,-113.797,-78.184,167.954,38.639,157.228
C00612=1035.332,-113.547,-78.194,167.957,38.638,157.228
C00613=1035.338,-113.297,-78.202,167.959,38.637,157.228
C00614=1035.344,-113.048,-78.212,167.962,38.636,157.227
C00615=1035.350,-112.798,-78.221,167.964,38.635,157.227
C00616=1035.356,-112.548,-78.231,167.967,38.634,157.227
C00617=1035.362,-112.298,-78.240,167.970,38.632,157.227
C00618=1035.368,-112.049,-78.250,167.972,38.632,157.227
C00619=1035.374,-111.799,-78.259,167.975,38.631,157.227
C00620=1035.380,-111.549,-78.268,167.978,38.630,157.227
C00621=1035.386,-111.299,-78.278,167.981,38.628,157.227
C00622=1035.392,-111.049,-78.287,167.984,38.628,157.227
C00623=1035.398,-110.800,-78.296,167.987,38.627,157.226
C00624=1035.404,-110.550,-78.306,167.988,38.625,157.226
C00625=1035.410,-110.301,-78.316,167.991,38.624,157.226
C00626=1035.416,-110.051,-78.325,167.994,38.624,157.226
C00627=1035.423,-109.801,-78.335,167.997,38.623,157.226
C00628=1035.429,-109.551,-78.344,168.000,38.621,157.226
C00629=1035.434,-109.302,-78.353,168.002,38.621,157.226
C00630=1035.441,-109.052,-78.363,168.005,38.620,157.226
C00631=1035.447,-108.802,-78.373,168.008,38.619,157.226
C00632=1035.453,-108.553,-78.382,168.010,38.617,157.225
C00633=1035.459,-108.303,-78.392,168.013,38.617,157.225
C00634=1035.465,-108.053,-78.401,168.015,38.616,157.225
C00635=1035.471,-107.803,-78.411,168.018,38.615,157.225
C00636=1035.477,-107.553,-78.421,168.021,38.613,157.225
C00637=1035.483,-107.303,-78.431,168.024,38.613,157.225
C00638=1035.489,-107.054,-78.440,168.027,38.612,157.225
C00639=1035.495,-106.804,-78.449,168.029,38.611,157.225
C00640=1035.501,-106.555,-78.459,168.032,38.610,157.225
C00641=1035.507,-106.305,-78.468,168.034,38.609,157.225
C00642=1035.513,-106.055,-78.479,168.037,38.608,157.224
C00643=1035.519,-105.805,-78.488,168.040,38.607,157.224
C00644=1035.525,-105.555,-78.498,168.042,38.606,157.224
C00645=1035.531,-105.305,-78.507,168.045,38.605,157.224
C00646=1035.537,-105.056,-78.517,168.048,38.605,157.224
C00647=1035.543,-104.806,-78.528,168.051,38.604,157.224
C00648=1035.549,-104.556,-78.537,168.053,38.603,157.224
C00649=1035.555,-104.306,-78.547,168.056,38.602,157.224
C00650=1035.561,-104.057,-78.556,168.059,38.601,157.224
C00651=1035.566,-103.807,-78.566,168.062,38.600,157.224
C00652=1035.572,-103.557,-78.576,168.064,38.599,157.224
C00653=1035.579,-103.308,-78.586,168.066,38.598,157.223
C00654=1035.585,-103.059,-78.596,168.069,38.597,157.223
C00655=1035.591,-102.808,-78.606,168.072,38.597,157.223
C00656=1035.597,-102.559,-78.615,168.075,38.596,157.223
C00657=1035.603,-102.309,-78.625,168.077,38.595,157.223
C00658=1035.609,-102.060,-78.635,168.080,38.594,157.223
C00659=1035.615,-101.810,-78.645,168.083,38.593,157.223
C00660=1035.621,-101.560,-78.655,168.086,38.592,157.223
C00661=1035.627,-101.310,-78.665,168.089,38.591,157.223
C00662=1035.633,-101.060,-78.675,168.090,38.590,157.223
C00663=1035.639,-100.811,-78.685,168.093,38.589,157.223
C00664=1035.646,-100.523,-78.696,168.096,38.589,157.223
C00665=1035.654,-100.236,-78.708,168.099,38.588,157.222
C00666=1035.660,-99.948,-78.719,168.103,38.587,157.222
C00667=1035.667,-99.662,-78.731,168.106,38.585,157.222
C00668=1035.673,-99.413,-78.740,168.109,38.585,157.222
C00669=1035.679,-99.162,-78.751,168.111,38.584,157.222
C00670=1035.686,-98.913,-78.761,168.114,38.583,157.222
C00671=1035.692,-98.663,-78.771,168.117,38.582,157.222
C00672=1035.698,-98.413,-78.781,168.119,38.581,157.222
C00673=1035.704,-98.163,-78.791,168.121,38.581,157.222
C00674=1035.710,-97.914,-78.801,168.124,38.580,157.222
C00675=1035.716,-97.664,-78.810,168.127,38.579,157.222
C00676=1035.722,-97.414,-78.821,168.130,38.578,157.222
C00677=1035.728,-97.165,-78.831,168.132,38.577,157.221
C00678=1035.734,-96.915,-78.842,168.135,38.577,157.221
C00679=1035.739,-96.665,-78.852,168.138,38.576,157.221
C00680=1035.746,-96.416,-78.862,168.140,38.576,157.221
C00681=1035.751,-96.166,-78.872,168.143,38.575,157.221
C00682=1035.758,-95.916,-78.883,168.146,38.574,157.221
C00683=1035.764,-95.666,-78.893,168.149,38.573,157.221
C00684=1035.770,-95.417,-78.903,168.151,38.572,157.221
C00685=1035.776,-95.166,-78.914,168.153,38.572,157.221
C00686=1035.782,-94.917,-78.924,168.156,38.571,157.221
C00687=1035.788,-94.667,-78.934,168.158,38.571,157.221
C00688=1035.794,-94.418,-78.944,168.161,38.570,157.221
C00689=1035.800,-94.168,-78.955,168.164,38.569,157.221
C00690=1035.805,-93.918,-78.965,168.167,38.568,157.221
C00691=1035.812,-93.668,-78.975,168.169,38.567,157.221
C00692=1035.818,-93.418,-78.986,168.172,38.567,157.221
C00693=1035.824,-93.169,-78.996,168.175,38.566,157.221
C00694=1035.830,-92.919,-79.007,168.177,38.566,157.220
C00695=1035.836,-92.670,-79.017,168.180,38.565,157.220
C00696=1035.842,-92.420,-79.027,168.183,38.564,157.220
C00697=1035.847,-92.170,-79.038,168.185,38.563,157.220
C00698=1035.855,-91.920,-79.049,168.188,38.563,157.220
C00699=1035.860,-91.670,-79.059,168.191,38.562,157.220
C00700=1035.866,-91.421,-79.069,168.193,38.561,157.220
C00701=1035.872,-91.172,-79.080,168.195,38.561,157.220
C00702=1035.878,-90.922,-79.090,168.198,38.560,157.220
C00703=1035.885,-90.672,-79.101,168.201,38.560,157.220
///RCONF 1,0,0,0,0,0,0,0,0,0,0,0,0,0,0,0,0,0,0,0,0,0,0,0
C00704=1035.890,-90.438,-79.110,168.203,38.559,157.220
C00705=1035.896,-90.205,-79.121,168.206,38.558,157.220
C00706=1035.902,-89.972,-79.130,168.208,38.557,157.220
C00707=1035.908,-89.739,-79.140,168.211,38.557,157.220
C00708=1035.913,-89.506,-79.150,168.213,38.556,157.220
C00709=1035.919,-89.272,-79.160,168.216,38.556,157.220
C00710=1035.924,-89.039,-79.170,168.218,38.555,157.220
C00711=1035.930,-88.806,-79.179,168.221,38.555,157.220
C00712=1035.936,-88.556,-79.190,168.224,38.554,157.219
C00713=1035.942,-88.307,-79.200,168.226,38.553,157.219
C00714=1035.948,-88.058,-79.211,168.229,38.552,157.219
C00715=1035.954,-87.807,-79.221,168.231,38.551,157.219
C00716=1035.961,-87.558,-79.232,168.234,38.551,157.219
C00717=1035.966,-87.308,-79.243,168.236,38.550,157.219
C00718=1035.973,-87.058,-79.254,168.239,38.550,157.219
C00719=1035.979,-86.809,-79.264,168.241,38.549,157.219
C00720=1035.985,-86.559,-79.274,168.244,38.548,157.219
C00721=1035.991,-86.309,-79.285,168.247,38.548,157.219
C00722=1035.997,-86.059,-79.296,168.249,38.547,157.219
C00723=1036.003,-85.810,-79.307,168.252,38.546,157.219
C00724=1036.010,-85.561,-79.317,168.255,38.545,157.219
C00725=1036.016,-85.310,-79.328,168.257,38.545,157.219
C00726=1036.022,-85.061,-79.339,168.260,38.545,157.219
C00727=1036.028,-84.811,-79.349,168.263,38.544,157.219
C00728=1036.036,-84.493,-79.363,168.266,38.543,157.219
C00729=1036.044,-84.176,-79.376,168.270,38.542,157.219
C00730=1036.052,-83.858,-79.390,168.273,38.541,157.218
C00731=1036.059,-83.539,-79.404,168.276,38.540,157.218
C00732=1036.066,-83.290,-79.414,168.278,38.540,157.218
C00733=1036.072,-83.040,-79.425,168.281,38.539,157.218
C00734=1036.078,-82.791,-79.436,168.284,38.539,157.218
C00735=1036.085,-82.541,-79.447,168.286,38.538,157.218
C00736=1036.091,-82.291,-79.457,168.289,38.537,157.218
C00737=1036.097,-82.041,-79.469,168.292,38.537,157.218
C00738=1036.103,-81.792,-79.479,168.294,38.536,157.218
C00739=1036.109,-81.542,-79.490,168.297,38.535,157.218
C00740=1036.116,-81.292,-79.501,168.300,38.534,157.218
C00741=1036.122,-81.043,-79.511,168.302,38.534,157.218
C00742=1036.128,-80.793,-79.523,168.305,38.534,157.218
C00743=1036.134,-80.543,-79.534,168.308,38.533,157.218
C00744=1036.141,-80.293,-79.544,168.310,38.533,157.218
C00745=1036.147,-80.044,-79.555,168.313,38.532,157.218
C00746=1036.153,-79.794,-79.566,168.316,38.531,157.218
C00747=1036.159,-79.544,-79.577,168.318,38.531,157.218
C00748=1036.165,-79.295,-79.588,168.320,38.530,157.218
C00749=1036.172,-79.045,-79.599,168.323,38.529,157.218
C00750=1036.178,-78.796,-79.610,168.325,38.529,157.218
C00751=1036.184,-78.546,-79.622,168.328,38.528,157.217
C00752=1036.190,-78.296,-79.632,168.330,38.528,157.217
C00753=1036.196,-78.047,-79.643,168.333,38.527,157.217
C00754=1036.202,-77.797,-79.655,168.336,38.527,157.217
C00755=1036.208,-77.547,-79.665,168.338,38.526,157.217
C00756=1036.214,-77.298,-79.677,168.341,38.526,157.217
C00757=1036.220,-77.048,-79.688,168.344,38.525,157.217
C00758=1036.226,-76.798,-79.699,168.346,38.525,157.217
C00759=1036.232,-76.548,-79.710,168.349,38.525,157.217
C00760=1036.239,-76.298,-79.722,168.351,38.524,157.217
C00761=1036.245,-76.050,-79.733,168.354,38.524,157.217
C00762=1036.252,-75.799,-79.744,168.357,38.523,157.217
C00763=1036.257,-75.550,-79.755,168.359,38.523,157.217
C00764=1036.264,-75.300,-79.766,168.362,38.522,157.217
C00765=1036.270,-75.051,-79.778,168.364,38.522,157.217
C00766=1036.276,-74.801,-79.789,168.367,38.521,157.217
C00767=1036.282,-74.551,-79.800,168.370,38.521,157.217
C00768=1036.288,-74.301,-79.811,168.372,38.520,157.217
C00769=1036.294,-74.052,-79.823,168.375,38.520,157.217
C00770=1036.301,-73.802,-79.834,168.377,38.519,157.217
C00771=1036.306,-73.552,-79.845,168.380,38.519,157.217
C00772=1036.312,-73.303,-79.857,168.383,38.519,157.217
C00773=1036.318,-73.053,-79.868,168.385,38.518,157.217
C00774=1036.325,-72.804,-79.880,168.388,38.518,157.217
C00775=1036.330,-72.554,-79.891,168.390,38.518,157.217
C00776=1036.337,-72.304,-79.902,168.393,38.517,157.217
C00777=1036.342,-72.055,-79.914,168.395,38.517,157.217
C00778=1036.348,-71.804,-79.926,168.398,38.517,157.217
C00779=1036.354,-71.556,-79.937,168.400,38.516,157.217
C00780=1036.361,-71.305,-79.948,168.402,38.516,157.217
C00781=1036.367,-71.057,-79.960,168.405,38.516,157.217
C00782=1036.372,-70.806,-79.972,168.407,38.515,157.217
C00783=1036.379,-70.556,-79.984,168.410,38.515,157.217
C00784=1036.385,-70.307,-79.995,168.412,38.515,157.217
C00785=1036.391,-70.057,-80.006,168.415,38.514,157.217
C00786=1036.397,-69.808,-80.018,168.417,38.514,157.217
C00787=1036.403,-69.557,-80.029,168.420,38.514,157.217
C00788=1036.409,-69.309,-80.041,168.422,38.513,157.217
C00789=1036.415,-69.059,-80.053,168.425,38.513,157.217
C00790=1036.422,-68.809,-80.064,168.428,38.512,157.217
C00791=1036.427,-68.560,-80.076,168.430,38.512,157.217
C00792=1036.434,-68.277,-80.089,168.433,38.512,157.217
C00793=1036.441,-67.994,-80.103,168.436,38.511,157.217
C00794=1036.448,-67.711,-80.116,168.439,38.511,157.217
C00795=1036.455,-67.428,-80.129,168.442,38.510,157.217
C00796=1036.461,-67.179,-80.141,168.444,38.510,157.217
C00797=1036.468,-66.928,-80.152,168.447,38.509,157.217
C00798=1036.474,-66.680,-80.164,168.449,38.509,157.217
C00799=1036.479,-66.429,-80.175,168.452,38.509,157.217
C00800=1036.485,-66.180,-80.187,168.454,38.508,157.217
C00801=1036.492,-65.931,-80.199,168.457,38.508,157.217
C00802=1036.498,-65.680,-80.210,168.459,38.508,157.217
C00803=1036.504,-65.431,-80.222,168.462,38.507,157.217
C00804=1036.510,-65.182,-80.234,168.465,38.507,157.217
C00805=1036.517,-64.931,-80.246,168.467,38.507,157.217
C00806=1036.523,-64.682,-80.257,168.470,38.506,157.217
C00807=1036.529,-64.433,-80.270,168.472,38.506,157.217
C00808=1036.535,-64.183,-80.281,168.475,38.506,157.217
C00809=1036.542,-63.933,-80.293,168.477,38.506,157.217
C00810=1036.548,-63.684,-80.304,168.480,38.505,157.217
C00811=1036.553,-63.434,-80.316,168.482,38.505,157.217
C00812=1036.560,-63.184,-80.328,168.485,38.505,157.217
C00813=1036.567,-62.934,-80.340,168.487,38.504,157.217
C00814=1036.572,-62.685,-80.352,168.490,38.504,157.217
C00815=1036.578,-62.435,-80.364,168.492,38.504,157.217
C00816=1036.585,-62.185,-80.376,168.495,38.504,157.217
C00817=1036.591,-61.937,-80.387,168.497,38.503,157.217
C00818=1036.597,-61.687,-80.400,168.500,38.503,157.217
C00819=1036.603,-61.437,-80.411,168.503,38.503,157.217
C00820=1036.610,-61.187,-80.423,168.505,38.502,157.217
C00821=1036.616,-60.937,-80.436,168.508,38.502,157.217
C00822=1036.622,-60.688,-80.447,168.510,38.502,157.217
C00823=1036.628,-60.438,-80.458,168.513,38.501,157.217
C00824=1036.635,-60.188,-80.470,168.515,38.501,157.217
C00825=1036.641,-59.939,-80.483,168.518,38.501,157.217
C00826=1036.647,-59.689,-80.495,168.520,38.500,157.217
C00827=1036.653,-59.440,-80.506,168.523,38.500,157.217
C00828=1036.659,-59.190,-80.519,168.525,38.500,157.217
C00829=1036.666,-58.940,-80.530,168.528,38.499,157.217
C00830=1036.672,-58.690,-80.542,168.530,38.499,157.217
C00831=1036.678,-58.441,-80.555,168.533,38.498,157.217
C00832=1036.684,-58.192,-80.566,168.535,38.498,157.217
C00833=1036.691,-57.942,-80.578,168.538,38.498,157.217
C00834=1036.697,-57.692,-80.591,168.540,38.498,157.217
C00835=1036.703,-57.443,-80.603,168.543,38.497,157.217
C00836=1036.710,-57.193,-80.615,168.545,38.497,157.217
C00837=1036.717,-56.944,-80.627,168.548,38.497,157.217
C00838=1036.723,-56.694,-80.639,168.550,38.497,157.217
C00839=1036.728,-56.444,-80.650,168.553,38.496,157.217
C00840=1036.735,-56.195,-80.662,168.555,38.496,157.217
C00841=1036.741,-55.945,-80.675,168.558,38.496,157.217
C00842=1036.748,-55.695,-80.687,168.560,38.495,157.217
C00843=1036.754,-55.446,-80.699,168.563,38.495,157.217
C00844=1036.760,-55.196,-80.711,168.565,38.495,157.217
C00845=1036.767,-54.946,-80.723,168.568,38.495,157.217
C00846=1036.773,-54.697,-80.735,168.570,38.494,157.217
C00847=1036.779,-54.447,-80.748,168.573,38.494,157.217
C00848=1036.786,-54.197,-80.760,168.575,38.494,157.217
C00849=1036.792,-53.947,-80.772,168.578,38.493,157.217
C00850=1036.798,-53.698,-80.784,168.579,38.493,157.217
C00851=1036.805,-53.449,-80.796,168.583,38.493,157.217
C00852=1036.810,-53.199,-80.808,168.585,38.492,157.217
C00853=1036.817,-52.950,-80.821,168.588,38.492,157.217
C00854=1036.824,-52.700,-80.833,168.589,38.492,157.217
C00855=1036.830,-52.450,-80.845,168.592,38.491,157.217
C00856=1036.838,-52.169,-80.859,168.595,38.491,157.217
C00857=1036.845,-51.887,-80.873,168.598,38.491,157.217
C00858=1036.852,-51.605,-80.887,168.600,38.490,157.217
C00859=1036.859,-51.324,-80.900,168.603,38.490,157.217
C00860=1036.866,-51.075,-80.913,168.606,38.490,157.217
C00861=1036.872,-50.825,-80.925,168.608,38.490,157.217
C00862=1036.878,-50.576,-80.937,168.611,38.489,157.217
C00863=1036.885,-50.326,-80.949,168.613,38.489,157.217
C00864=1036.891,-50.076,-80.962,168.615,38.489,157.217
C00865=1036.897,-49.826,-80.974,168.618,38.489,157.217
C00866=1036.903,-49.577,-80.988,168.620,38.489,157.217
C00867=1036.909,-49.327,-81.000,168.623,38.488,157.217
C00868=1036.915,-49.077,-81.012,168.625,38.488,157.217
C00869=1036.921,-48.828,-81.025,168.627,38.488,157.217
C00870=1036.928,-48.579,-81.037,168.631,38.488,157.217
C00871=1036.934,-48.329,-81.050,168.633,38.488,157.217
C00872=1036.940,-48.079,-81.062,168.636,38.488,157.217
C00873=1036.946,-47.830,-81.076,168.638,38.488,157.217
C00874=1036.953,-47.580,-81.088,168.641,38.488,157.217
C00875=1036.959,-47.330,-81.100,168.643,38.487,157.217
C00876=1036.965,-47.081,-81.113,168.645,38.487,157.217
C00877=1036.972,-46.831,-81.125,168.648,38.487,157.217
C00878=1036.978,-46.581,-81.138,168.650,38.487,157.217
C00879=1036.984,-46.332,-81.151,168.653,38.487,157.218
C00880=1036.990,-46.082,-81.164,168.655,38.487,157.218
C00881=1036.996,-45.833,-81.176,168.657,38.487,157.218
C00882=1037.003,-45.583,-81.189,168.660,38.487,157.218
C00883=1037.008,-45.334,-81.202,168.662,38.487,157.218
C00884=1037.014,-45.084,-81.214,168.665,38.486,157.218
C00885=1037.021,-44.835,-81.227,168.667,38.486,157.218
C00886=1037.027,-44.585,-81.239,168.669,38.486,157.218
C00887=1037.033,-44.336,-81.253,168.672,38.486,157.218
C00888=1037.040,-44.085,-81.266,168.674,38.486,157.218
C00889=1037.047,-43.836,-81.278,168.677,38.486,157.218
C00890=1037.053,-43.586,-81.291,168.679,38.486,157.218
C00891=1037.059,-43.336,-81.303,168.681,38.486,157.218
C00892=1037.065,-43.087,-81.317,168.684,38.485,157.218
C00893=1037.072,-42.837,-81.329,168.686,38.485,157.218
C00894=1037.078,-42.588,-81.342,168.689,38.485,157.218
C00895=1037.084,-42.338,-81.354,168.691,38.486,157.218
C00896=1037.090,-42.089,-81.368,168.693,38.486,157.218
C00897=1037.097,-41.839,-81.380,168.696,38.485,157.218
C00898=1037.103,-41.590,-81.393,168.698,38.485,157.218
C00899=1037.109,-41.340,-81.406,168.701,38.485,157.218
C00900=1037.115,-41.090,-81.419,168.703,38.485,157.218
C00901=1037.121,-40.840,-81.432,168.705,38.485,157.218
C00902=1037.128,-40.592,-81.444,168.708,38.485,157.218
C00903=1037.134,-40.342,-81.457,168.710,38.485,157.218
C00904=1037.141,-40.092,-81.470,168.713,38.485,157.218
C00905=1037.147,-39.842,-81.484,168.715,38.484,157.218
C00906=1037.154,-39.593,-81.496,168.717,38.484,157.218
C00907=1037.160,-39.344,-81.509,168.720,38.484,157.219
C00908=1037.166,-39.094,-81.522,168.722,38.484,157.219
C00909=1037.172,-38.844,-81.535,168.725,38.484,157.219
C00910=1037.179,-38.594,-81.548,168.727,38.484,157.219
C00911=1037.185,-38.345,-81.561,168.729,38.484,157.219
C00912=1037.191,-38.095,-81.574,168.732,38.484,157.219
C00913=1037.197,-37.846,-81.588,168.734,38.483,157.219
C00914=1037.203,-37.596,-81.600,168.736,38.484,157.219
C00915=1037.210,-37.347,-81.613,168.739,38.484,157.219
C00916=1037.216,-37.097,-81.627,168.741,38.484,157.219
C00917=1037.222,-36.847,-81.640,168.743,38.484,157.219
C00918=1037.228,-36.598,-81.653,168.747,38.483,157.219
C00919=1037.235,-36.349,-81.666,168.749,38.484,157.219
C00920=1037.242,-36.067,-81.681,168.752,38.484,157.219
C00921=1037.249,-35.786,-81.696,168.754,38.484,157.219
C00922=1037.256,-35.505,-81.710,168.757,38.484,157.219
C00923=1037.262,-35.224,-81.725,168.759,38.484,157.219
C00924=1037.269,-34.974,-81.739,168.762,38.484,157.219
C00925=1037.275,-34.724,-81.752,168.764,38.484,157.219
C00926=1037.282,-34.475,-81.766,168.766,38.484,157.219
C00927=1037.288,-34.226,-81.779,168.769,38.484,157.219
C00928=1037.294,-33.976,-81.791,168.771,38.484,157.220
C00929=1037.300,-33.727,-81.805,168.773,38.483,157.220
C00930=1037.307,-33.477,-81.818,168.776,38.484,157.220
C00931=1037.313,-33.227,-81.832,168.778,38.484,157.220
C00932=1037.319,-32.978,-81.845,168.780,38.484,157.220
C00933=1037.326,-32.728,-81.858,168.783,38.484,157.220
C00934=1037.332,-32.478,-81.871,168.785,38.483,157.220
C00935=1037.338,-32.229,-81.884,168.787,38.484,157.220
C00936=1037.344,-31.980,-81.898,168.790,38.484,157.220
C00937=1037.351,-31.730,-81.911,168.792,38.484,157.220
C00938=1037.357,-31.481,-81.924,168.794,38.484,157.220
C00939=1037.364,-31.231,-81.938,168.797,38.484,157.220
C00940=1037.370,-30.981,-81.951,168.799,38.483,157.220
C00941=1037.377,-30.732,-81.965,168.801,38.484,157.220
C00942=1037.382,-30.482,-81.978,168.804,38.484,157.220
C00943=1037.389,-30.232,-81.991,168.806,38.484,157.220
C00944=1037.395,-29.983,-82.005,168.808,38.484,157.220
C00945=1037.401,-29.733,-82.018,168.810,38.484,157.220
C00946=1037.408,-29.483,-82.032,168.814,38.484,157.221
C00947=1037.414,-29.234,-82.045,168.816,38.484,157.221
C00948=1037.420,-28.985,-82.058,168.818,38.484,157.221
C00949=1037.427,-28.735,-82.072,168.821,38.484,157.221
C00950=1037.433,-28.486,-82.085,168.823,38.484,157.221
C00951=1037.439,-28.236,-82.098,168.825,38.483,157.221
C00952=1037.446,-27.986,-82.112,168.828,38.484,157.221
C00953=1037.453,-27.737,-82.125,168.830,38.484,157.221
C00954=1037.458,-27.488,-82.139,168.832,38.484,157.221
C00955=1037.465,-27.238,-82.153,168.835,38.484,157.221
C00956=1037.471,-26.988,-82.166,168.837,38.483,157.221
C00957=1037.478,-26.738,-82.180,168.839,38.484,157.221
C00958=1037.483,-26.489,-82.193,168.841,38.484,157.221
C00959=1037.490,-26.240,-82.207,168.844,38.484,157.221
C00960=1037.496,-25.990,-82.220,168.846,38.484,157.221
C00961=1037.502,-25.741,-82.235,168.848,38.484,157.221
C00962=1037.509,-25.491,-82.249,168.850,38.484,157.221
C00963=1037.515,-25.241,-82.262,168.853,38.485,157.222
C00964=1037.521,-24.992,-82.276,168.855,38.484,157.222
C00965=1037.527,-24.742,-82.289,168.857,38.484,157.222
C00966=1037.534,-24.493,-82.303,168.859,38.485,157.222
C00967=1037.539,-24.243,-82.316,168.862,38.485,157.222
C00968=1037.546,-23.994,-82.331,168.865,38.485,157.222
C00969=1037.552,-23.744,-82.344,168.867,38.485,157.222
C00970=1037.559,-23.494,-82.358,168.869,38.485,157.222
C00971=1037.565,-23.245,-82.372,168.872,38.486,157.222
C00972=1037.572,-22.995,-82.385,168.874,38.486,157.222
C00973=1037.577,-22.746,-82.400,168.876,38.485,157.222
C00974=1037.584,-22.497,-82.413,168.878,38.486,157.222
C00975=1037.590,-22.247,-82.427,168.881,38.486,157.222
C00976=1037.596,-21.997,-82.441,168.883,38.486,157.222
C00977=1037.603,-21.748,-82.455,168.885,38.486,157.223
C00978=1037.609,-21.499,-82.468,168.887,38.486,157.223
C00979=1037.615,-21.248,-82.482,168.890,38.486,157.223
C00980=1037.621,-20.999,-82.496,168.892,38.487,157.223
C00981=1037.629,-20.750,-82.510,168.894,38.486,157.223
C00982=1037.634,-20.500,-82.524,168.896,38.486,157.223
C00983=1037.641,-20.250,-82.538,168.898,38.487,157.223
C00984=1037.648,-19.969,-82.553,168.901,38.487,157.223
C00985=1037.655,-19.687,-82.569,168.904,38.487,157.223
C00986=1037.663,-19.405,-82.585,168.907,38.487,157.223
C00987=1037.669,-19.124,-82.601,168.910,38.487,157.223
C00988=1037.676,-18.873,-82.615,168.912,38.487,157.223
C00989=1037.682,-18.624,-82.628,168.914,38.487,157.223
C00990=1037.688,-18.374,-82.643,168.916,38.487,157.223
C00991=1037.694,-18.125,-82.656,168.919,38.487,157.223
C00992=1037.701,-17.875,-82.670,168.921,38.488,157.224
C00993=1037.707,-17.626,-82.684,168.923,38.488,157.224
C00994=1037.714,-17.376,-82.698,168.925,38.487,157.224
C00995=1037.720,-17.128,-82.712,168.927,38.488,157.224
C00996=1037.726,-16.877,-82.726,168.930,38.488,157.224
C00997=1037.733,-16.627,-82.740,168.932,38.488,157.224
C00998=1037.739,-16.378,-82.755,168.934,38.488,157.224
C00999=1037.746,-16.128,-82.768,168.936,38.488,157.224
C01000=1037.752,-15.880,-82.782,168.939,38.488,157.224
C01001=1037.758,-15.630,-82.796,168.941,38.489,157.224
C01002=1037.765,-15.380,-82.810,168.943,38.488,157.224
C01003=1037.771,-15.131,-82.825,168.945,38.489,157.224
C01004=1037.777,-14.880,-82.839,168.947,38.489,157.224
C01005=1037.784,-14.632,-82.853,168.951,38.489,157.225
C01006=1037.790,-14.382,-82.868,168.953,38.489,157.225
C01007=1037.796,-14.133,-82.881,168.955,38.490,157.225
C01008=1037.803,-13.883,-82.896,168.957,38.490,157.225
C01009=1037.808,-13.634,-82.910,168.959,38.490,157.225
C01010=1037.815,-13.384,-82.924,168.961,38.490,157.225
C01011=1037.821,-13.134,-82.938,168.964,38.490,157.225
C01012=1037.827,-12.885,-82.953,168.966,38.491,157.225
C01013=1037.834,-12.635,-82.967,168.968,38.491,157.225
C01014=1037.840,-12.386,-82.981,168.970,38.491,157.225
C01015=1037.846,-12.136,-82.996,168.972,38.491,157.225
C01016=1037.853,-11.886,-83.010,168.974,38.491,157.225
C01017=1037.859,-11.637,-83.024,168.977,38.491,157.226
C01018=1037.865,-11.388,-83.039,168.979,38.492,157.226
C01019=1037.871,-11.139,-83.053,168.981,38.492,157.226
C01020=1037.878,-10.889,-83.068,168.984,38.492,157.226
C01021=1037.884,-10.639,-83.081,168.986,38.492,157.226
C01022=1037.890,-10.390,-83.096,168.988,38.493,157.226
C01023=1037.897,-10.140,-83.111,168.991,38.493,157.226
C01024=1037.903,-9.890,-83.124,168.993,38.493,157.226
C01025=1037.909,-9.641,-83.139,168.995,38.493,157.226
C01026=1037.916,-9.392,-83.154,168.997,38.494,157.226
C01027=1037.923,-9.142,-83.168,168.999,38.493,157.226
C01028=1037.928,-8.893,-83.182,169.001,38.494,157.227
C01029=1037.935,-8.643,-83.197,169.004,38.494,157.227
C01030=1037.942,-8.394,-83.211,169.006,38.494,157.227
C01031=1037.947,-8.144,-83.225,169.008,38.494,157.227
C01032=1037.954,-7.895,-83.240,169.010,38.494,157.227
C01033=1037.960,-7.645,-83.255,169.012,38.495,157.227
C01034=1037.966,-7.396,-83.269,169.014,38.495,157.227
C01035=1037.972,-7.146,-83.283,169.017,38.495,157.227
C01036=1037.979,-6.896,-83.298,169.019,38.495,157.227
C01037=1037.985,-6.648,-83.312,169.022,38.496,157.227
C01038=1037.992,-6.398,-83.327,169.024,38.495,157.227
C01039=1037.998,-6.148,-83.342,169.026,38.496,157.227
C01040=1038.005,-5.898,-83.356,169.028,38.496,157.227
C01041=1038.011,-5.649,-83.370,169.030,38.496,157.228
C01042=1038.017,-5.400,-83.385,169.033,38.496,157.228
C01043=1038.024,-5.150,-83.400,169.035,38.497,157.228
C01044=1038.031,-4.901,-83.415,169.037,38.497,157.228
C01045=1038.036,-4.651,-83.428,169.039,38.497,157.228
C01046=1038.043,-4.402,-83.443,169.041,38.497,157.228
C01047=1038.050,-4.152,-83.458,169.043,38.497,157.228
C01048=1038.057,-3.869,-83.474,169.046,38.498,157.228
C01049=1038.064,-3.586,-83.491,169.048,38.497,157.228
C01050=1038.070,-3.302,-83.508,169.051,38.498,157.228
C01051=1038.078,-3.018,-83.525,169.054,38.499,157.229
C01052=1038.084,-2.769,-83.539,169.056,38.499,157.229
C01053=1038.090,-2.519,-83.554,169.058,38.499,157.229
C01054=1038.097,-2.270,-83.569,169.060,38.499,157.229
C01055=1038.103,-2.020,-83.584,169.062,38.500,157.229
C01056=1038.109,-1.771,-83.599,169.064,38.500,157.229
C01057=1038.115,-1.521,-83.614,169.066,38.500,157.229
C01058=1038.122,-1.272,-83.629,169.069,38.501,157.229
C01059=1038.128,-1.022,-83.644,169.071,38.501,157.229
C01060=1038.134,-0.773,-83.658,169.073,38.501,157.229
C01061=1038.140,-0.523,-83.673,169.075,38.501,157.230
C01062=1038.147,-0.274,-83.688,169.077,38.502,157.230
C01063=1038.153,-0.024,-83.703,169.080,38.502,157.230
C01064=1038.159,0.225,-83.718,169.082,38.502,157.230
C01065=1038.165,0.474,-83.733,169.084,38.503,157.230
C01066=1038.171,0.724,-83.748,169.086,38.503,157.230
C01067=1038.178,0.973,-83.763,169.088,38.503,157.230
C01068=1038.185,1.223,-83.778,169.090,38.504,157.230
C01069=1038.190,1.472,-83.793,169.092,38.504,157.230
C01070=1038.197,1.721,-83.808,169.095,38.504,157.230
C01071=1038.203,1.971,-83.823,169.097,38.505,157.231
C01072=1038.209,2.221,-83.838,169.099,38.505,157.231
C01073=1038.216,2.470,-83.853,169.101,38.505,157.231
C01074=1038.222,2.720,-83.867,169.104,38.506,157.231
C01075=1038.227,2.969,-83.883,169.106,38.506,157.231
C01076=1038.234,3.218,-83.898,169.108,38.506,157.231
C01077=1038.240,3.468,-83.913,169.110,38.507,157.231
C01078=1038.247,3.718,-83.928,169.112,38.507,157.231
C01079=1038.253,3.967,-83.943,169.114,38.507,157.231
C01080=1038.259,4.217,-83.958,169.116,38.508,157.232
C01081=1038.266,4.467,-83.973,169.118,38.508,157.232
C01082=1038.272,4.715,-83.988,169.120,38.508,157.232
C01083=1038.278,4.965,-84.003,169.123,38.509,157.232
C01084=1038.285,5.214,-84.018,169.125,38.508,157.232
C01085=1038.291,5.464,-84.033,169.127,38.509,157.232
C01086=1038.298,5.713,-84.049,169.129,38.509,157.232
C01087=1038.304,5.963,-84.064,169.132,38.509,157.232
C01088=1038.311,6.212,-84.079,169.134,38.510,157.232
C01089=1038.317,6.462,-84.094,169.136,38.510,157.232
C01090=1038.324,6.711,-84.109,169.138,38.510,157.233
C01091=1038.329,6.960,-84.125,169.140,38.511,157.233
C01092=1038.335,7.210,-84.139,169.142,38.511,157.233
C01093=1038.341,7.460,-84.154,169.144,38.511,157.233
C01094=1038.348,7.709,-84.170,169.146,38.511,157.233
C01095=1038.355,7.958,-84.185,169.148,38.512,157.233
C01096=1038.361,8.208,-84.200,169.150,38.512,157.233
C01097=1038.368,8.457,-84.216,169.152,38.512,157.233
C01098=1038.374,8.707,-84.231,169.154,38.513,157.233
C01099=1038.380,8.956,-84.246,169.157,38.513,157.233
C01100=1038.387,9.206,-84.260,169.160,38.513,157.234
C01101=1038.393,9.455,-84.276,169.162,38.514,157.234
C01102=1038.399,9.705,-84.292,169.164,38.514,157.234
C01103=1038.406,9.954,-84.307,169.166,38.514,157.234
C01104=1038.412,10.204,-84.322,169.168,38.514,157.234
C01105=1038.419,10.453,-84.337,169.170,38.515,157.234
C01106=1038.425,10.702,-84.353,169.172,38.515,157.234
C01107=1038.432,10.952,-84.368,169.174,38.515,157.234
C01108=1038.438,11.202,-84.383,169.176,38.516,157.234
C01109=1038.445,11.451,-84.398,169.178,38.516,157.234
C01110=1038.451,11.700,-84.413,169.180,38.516,157.235
C01111=1038.458,11.949,-84.429,169.183,38.517,157.235
C01112=1038.464,12.236,-84.447,169.186,38.516,157.235
C01113=1038.472,12.521,-84.464,169.188,38.517,157.235
C01114=1038.479,12.806,-84.482,169.190,38.518,157.235
C01115=1038.487,13.091,-84.500,169.193,38.517,157.235
C01116=1038.493,13.341,-84.515,169.195,38.518,157.235
C01117=1038.500,13.590,-84.530,169.197,38.518,157.235
C01118=1038.506,13.840,-84.545,169.199,38.518,157.235
C01119=1038.513,14.089,-84.561,169.201,38.519,157.236
C01120=1038.519,14.339,-84.576,169.203,38.519,157.236
C01121=1038.525,14.588,-84.592,169.205,38.519,157.236
C01122=1038.532,14.837,-84.607,169.207,38.520,157.236
C01123=1038.538,15.087,-84.623,169.210,38.520,157.236
C01124=1038.544,15.336,-84.638,169.212,38.521,157.236
C01125=1038.551,15.585,-84.654,169.214,38.521,157.236
C01126=1038.556,15.835,-84.669,169.216,38.521,157.236
C01127=1038.563,16.084,-84.685,169.218,38.522,157.236
C01128=1038.569,16.334,-84.701,169.220,38.522,157.237
C01129=1038.575,16.583,-84.716,169.222,38.522,157.237
C01130=1038.582,16.832,-84.732,169.224,38.523,157.237
C01131=1038.588,17.082,-84.748,169.226,38.523,157.237
C01132=1038.594,17.331,-84.763,169.228,38.523,157.237
C01133=1038.602,17.581,-84.779,169.230,38.524,157.237
C01134=1038.607,17.831,-84.795,169.233,38.524,157.237
C01135=1038.614,18.080,-84.810,169.235,38.525,157.237
C01136=1038.620,18.329,-84.827,169.237,38.525,157.237
C01137=1038.626,18.579,-84.842,169.239,38.525,157.238
C01138=1038.633,18.828,-84.857,169.241,38.526,157.238
C01139=1038.639,19.077,-84.874,169.243,38.526,157.238
C01140=1038.645,19.327,-84.888,169.245,38.526,157.238
C01141=1038.651,19.576,-84.905,169.247,38.527,157.238
C01142=1038.658,19.825,-84.920,169.249,38.527,157.238
C01143=1038.665,20.075,-84.936,169.251,38.527,157.238
C01144=1038.671,20.325,-84.952,169.253,38.528,157.238
C01145=1038.678,20.574,-84.968,169.256,38.528,157.239
C01146=1038.684,20.824,-84.984,169.258,38.529,157.239
C01147=1038.690,21.073,-85.000,169.260,38.529,157.239
C01148=1038.696,21.323,-85.015,169.262,38.529,157.239
C01149=1038.702,21.572,-85.031,169.264,38.530,157.239
C01150=1038.709,21.821,-85.047,169.266,38.530,157.239
C01151=1038.715,22.070,-85.063,169.268,38.531,157.239
C01152=1038.722,22.320,-85.079,169.270,38.531,157.239
C01153=1038.727,22.570,-85.095,169.272,38.531,157.239
C01154=1038.734,22.819,-85.110,169.274,38.532,157.240
C01155=1038.740,23.068,-85.127,169.277,38.532,157.240
C01156=1038.747,23.317,-85.142,169.279,38.533,157.240
C01157=1038.753,23.567,-85.159,169.281,38.533,157.240
C01158=1038.759,23.816,-85.174,169.283,38.533,157.240
C01159=1038.766,24.067,-85.190,169.285,38.534,157.240
C01160=1038.772,24.316,-85.206,169.287,38.535,157.240
C01161=1038.778,24.565,-85.222,169.289,38.534,157.240
C01162=1038.785,24.814,-85.238,169.290,38.535,157.241
C01163=1038.791,25.063,-85.254,169.292,38.536,157.241
C01164=1038.798,25.313,-85.271,169.294,38.536,157.241
C01165=1038.804,25.562,-85.286,169.297,38.536,157.241
C01166=1038.810,25.812,-85.303,169.299,38.536,157.241
C01167=1038.817,26.061,-85.318,169.301,38.537,157.241
C01168=1038.823,26.310,-85.335,169.303,38.538,157.241
C01169=1038.830,26.560,-85.350,169.305,38.538,157.241
C01170=1038.836,26.810,-85.366,169.307,38.538,157.241
C01171=1038.842,27.059,-85.382,169.309,38.539,157.242
C01172=1038.848,27.308,-85.398,169.311,38.539,157.242
C01173=1038.854,27.558,-85.414,169.313,38.540,157.242
C01174=1038.862,27.807,-85.430,169.315,38.540,157.242
C01175=1038.868,28.057,-85.447,169.318,38.540,157.242
C01176=1038.875,28.343,-85.465,169.320,38.541,157.242
C01177=1038.882,28.629,-85.484,169.323,38.541,157.242
C01178=1038.889,28.917,-85.503,169.325,38.542,157.243
C01179=1038.897,29.203,-85.521,169.327,38.542,157.243
C01180=1038.903,29.453,-85.538,169.329,38.543,157.243
C01181=1038.909,29.702,-85.554,169.331,38.543,157.243
C01182=1038.915,29.951,-85.570,169.333,38.544,157.243
C01183=1038.922,30.201,-85.586,169.336,38.544,157.243
C01184=1038.928,30.450,-85.602,169.338,38.544,157.243
C01185=1038.934,30.700,-85.619,169.340,38.545,157.243
C01186=1038.941,30.948,-85.635,169.342,38.545,157.244
C01187=1038.947,31.198,-85.652,169.343,38.546,157.244
C01188=1038.953,31.448,-85.668,169.345,38.546,157.244
C01189=1038.959,31.697,-85.684,169.347,38.547,157.244
C01190=1038.965,31.946,-85.700,169.349,38.547,157.244
C01191=1038.972,32.196,-85.716,169.351,38.547,157.244
C01192=1038.978,32.445,-85.733,169.353,38.548,157.244
C01193=1038.985,32.694,-85.750,169.356,38.548,157.245
C01194=1038.991,32.944,-85.766,169.358,38.549,157.245
C01195=1038.997,33.193,-85.783,169.360,38.549,157.245
C01196=1039.004,33.442,-85.798,169.362,38.550,157.245
C01197=1039.010,33.693,-85.815,169.364,38.551,157.245
C01198=1039.016,33.942,-85.831,169.366,38.550,157.245
C01199=1039.023,34.191,-85.848,169.368,38.551,157.245
C01200=1039.029,34.440,-85.864,169.370,38.552,157.245
C01201=1039.036,34.690,-85.880,169.372,38.552,157.246
C01202=1039.042,34.939,-85.897,169.375,38.553,157.246
C01203=1039.048,35.188,-85.914,169.376,38.553,157.246
C01204=1039.055,35.438,-85.930,169.378,38.553,157.246
C01205=1039.061,35.687,-85.946,169.380,38.554,157.246
C01206=1039.067,35.936,-85.962,169.382,38.554,157.246
C01207=1039.074,36.186,-85.979,169.384,38.555,157.246
C01208=1039.080,36.435,-85.996,169.386,38.555,157.246
C01209=1039.087,36.685,-86.012,169.388,38.556,157.247
C01210=1039.093,36.934,-86.029,169.390,38.556,157.247
C01211=1039.100,37.183,-86.045,169.392,38.556,157.247
C01212=1039.106,37.433,-86.062,169.395,38.557,157.247
C01213=1039.112,37.682,-86.078,169.397,38.557,157.247
C01214=1039.118,37.931,-86.095,169.399,38.558,157.247
C01215=1039.125,38.181,-86.111,169.401,38.558,157.247
C01216=1039.131,38.430,-86.128,169.402,38.559,157.248
C01217=1039.137,38.679,-86.145,169.404,38.559,157.248
C01218=1039.144,38.929,-86.161,169.406,38.560,157.248
C01219=1039.149,39.178,-86.179,169.408,38.560,157.248
C01220=1039.156,39.428,-86.195,169.411,38.561,157.248
C01221=1039.162,39.678,-86.212,169.413,38.561,157.248
C01222=1039.168,39.926,-86.229,169.415,38.561,157.248
C01223=1039.174,40.176,-86.245,169.417,38.562,157.248
C01224=1039.181,40.425,-86.262,169.419,38.563,157.249
C01225=1039.187,40.674,-86.279,169.421,38.563,157.249
C01226=1039.194,40.924,-86.296,169.422,38.564,157.249
C01227=1039.199,41.173,-86.312,169.424,38.564,157.249
C01228=1039.206,41.423,-86.330,169.426,38.565,157.249
C01229=1039.212,41.672,-86.346,169.429,38.565,157.249
C01230=1039.219,41.921,-86.363,169.431,38.566,157.249
C01231=1039.225,42.171,-86.379,169.433,38.566,157.250
C01232=1039.231,42.419,-86.396,169.435,38.567,157.250
C01233=1039.238,42.670,-86.413,169.437,38.567,157.250
C01234=1039.244,42.918,-86.430,169.439,38.567,157.250
C01235=1039.251,43.168,-86.447,169.441,38.568,157.250
C01236=1039.257,43.417,-86.464,169.442,38.568,157.250
C01237=1039.262,43.667,-86.480,169.444,38.569,157.250
C01238=1039.269,43.916,-86.498,169.446,38.569,157.251
C01239=1039.275,44.165,-86.514,169.449,38.571,157.251
C01240=1039.283,44.452,-86.534,169.451,38.571,157.251
C01241=1039.289,44.739,-86.554,169.453,38.572,157.251
C01242=1039.296,45.025,-86.573,169.455,38.572,157.251
C01243=1039.303,45.312,-86.593,169.458,38.573,157.251
C01244=1039.309,45.561,-86.609,169.459,38.573,157.252
C01245=1039.316,45.811,-86.627,169.461,38.574,157.252
C01246=1039.322,46.060,-86.644,169.464,38.574,157.252
C01247=1039.328,46.309,-86.660,169.466,38.576,157.252
C01248=1039.335,46.558,-86.678,169.468,38.576,157.252
C01249=1039.340,46.808,-86.695,169.470,38.577,157.252
C01250=1039.347,47.058,-86.712,169.472,38.577,157.253
C01251=1039.353,47.306,-86.729,169.474,38.578,157.253
C01252=1039.359,47.556,-86.747,169.475,38.578,157.253
C01253=1039.365,47.805,-86.764,169.478,38.579,157.253
C01254=1039.372,48.055,-86.781,169.480,38.579,157.253
C01255=1039.377,48.304,-86.798,169.482,38.580,157.253
C01256=1039.384,48.553,-86.815,169.484,38.580,157.253
C01257=1039.390,48.803,-86.832,169.486,38.581,157.254
C01258=1039.396,49.052,-86.850,169.488,38.581,157.254
C01259=1039.403,49.301,-86.867,169.489,38.582,157.254
C01260=1039.409,49.551,-86.884,169.491,38.583,157.254
C01261=1039.415,49.800,-86.901,169.494,38.583,157.254
C01262=1039.421,50.050,-86.918,169.496,38.584,157.254
C01263=1039.428,50.298,-86.935,169.498,38.584,157.254
C01264=1039.435,50.548,-86.952,169.500,38.585,157.255
C01265=1039.440,50.797,-86.970,169.502,38.585,157.255
C01266=1039.447,51.047,-86.987,169.503,38.586,157.255
C01267=1039.452,51.296,-87.004,169.505,38.586,157.255
C01268=1039.459,51.545,-87.022,169.507,38.587,157.255
C01269=1039.465,51.794,-87.038,169.510,38.587,157.255
C01270=1039.471,52.044,-87.056,169.512,38.588,157.255
C01271=1039.478,52.293,-87.073,169.514,38.588,157.256
C01272=1039.484,52.543,-87.090,169.516,38.589,157.256
C01273=1039.490,52.792,-87.108,169.518,38.590,157.256
C01274=1039.497,53.041,-87.125,169.519,38.590,157.256
C01275=1039.503,53.291,-87.142,169.521,38.591,157.256
C01276=1039.509,53.540,-87.160,169.523,38.591,157.256
C01277=1039.516,53.789,-87.177,169.526,38.592,157.257
C01278=1039.522,54.038,-87.194,169.528,38.592,157.257
C01279=1039.528,54.287,-87.212,169.530,38.593,157.257
C01280=1039.535,54.537,-87.229,169.532,38.593,157.257
C01281=1039.541,54.786,-87.246,169.534,38.594,157.257
C01282=1039.547,55.036,-87.264,169.535,38.594,157.257
C01283=1039.553,55.285,-87.281,169.537,38.595,157.257
C01284=1039.560,55.534,-87.298,169.539,38.595,157.258
C01285=1039.566,55.784,-87.316,169.542,38.596,157.258
C01286=1039.573,56.033,-87.333,169.544,38.597,157.258
C01287=1039.579,56.282,-87.351,169.546,38.596,157.258
C01288=1039.585,56.531,-87.368,169.548,38.597,157.258
C01289=1039.592,56.780,-87.385,169.550,38.597,157.258
C01290=1039.598,57.030,-87.403,169.551,38.598,157.258
C01291=1039.604,57.279,-87.420,169.553,38.599,157.258
C01292=1039.611,57.528,-87.437,169.555,38.599,157.259
C01293=1039.617,57.778,-87.455,169.557,38.600,157.259
C01294=1039.623,58.027,-87.472,169.560,38.600,157.259
C01295=1039.630,58.277,-87.490,169.562,38.601,157.259
C01296=1039.636,58.526,-87.507,169.564,38.601,157.259
C01297=1039.643,58.775,-87.524,169.566,38.602,157.259
C01298=1039.649,59.025,-87.542,169.567,38.602,157.259
C01299=1039.656,59.274,-87.560,169.569,38.603,157.260
C01300=1039.661,59.523,-87.577,169.571,38.603,157.260
C01301=1039.668,59.772,-87.595,169.573,38.604,157.260
C01302=1039.675,60.022,-87.612,169.576,38.604,157.260
C01303=1039.681,60.272,-87.630,169.578,38.605,157.260
C01304=1039.688,60.558,-87.650,169.580,38.606,157.260
C01305=1039.696,60.844,-87.670,169.582,38.606,157.261
C01306=1039.703,61.130,-87.690,169.584,38.607,157.261
C01307=1039.711,61.416,-87.710,169.586,38.607,157.261
C01308=1039.717,61.665,-87.728,169.588,38.608,157.261
C01309=1039.724,61.914,-87.745,169.590,38.608,157.261
C01310=1039.730,62.164,-87.763,169.593,38.609,157.261
C01311=1039.737,62.413,-87.781,169.595,38.609,157.261
C01312=1039.743,62.662,-87.798,169.597,38.609,157.261
C01313=1039.749,62.912,-87.816,169.599,38.610,157.262
C01314=1039.756,63.161,-87.833,169.601,38.610,157.262
C01315=1039.762,63.411,-87.851,169.603,38.611,157.262
C01316=1039.768,63.659,-87.869,169.604,38.611,157.262
C01317=1039.775,63.909,-87.887,169.606,38.612,157.262
C01318=1039.781,64.158,-87.904,169.608,38.612,157.262
C01319=1039.788,64.408,-87.922,169.611,38.613,157.262
C01320=1039.793,64.657,-87.940,169.613,38.613,157.263
C01321=1039.800,64.906,-87.957,169.615,38.614,157.263
C01322=1039.806,65.156,-87.975,169.617,38.614,157.263
C01323=1039.812,65.405,-87.993,169.618,38.615,157.263
C01324=1039.819,65.654,-88.011,169.620,38.616,157.263
C01325=1039.825,65.903,-88.029,169.622,38.616,157.263
C01326=1039.831,66.153,-88.047,169.625,38.617,157.264
C01327=1039.838,66.402,-88.065,169.627,38.618,157.264
C01328=1039.844,66.651,-88.082,169.629,38.618,157.264
C01329=1039.850,66.901,-88.100,169.630,38.619,157.264
C01330=1039.857,67.150,-88.118,169.632,38.619,157.264
C01331=1039.863,67.399,-88.136,169.634,38.620,157.264
C01332=1039.869,67.648,-88.154,169.636,38.620,157.265
C01333=1039.875,67.897,-88.173,169.638,38.621,157.265
C01334=1039.882,68.147,-88.190,169.641,38.621,157.265
C01335=1039.888,68.397,-88.208,169.643,38.622,157.265
C01336=1039.895,68.646,-88.227,169.644,38.623,157.265
C01337=1039.900,68.895,-88.244,169.646,38.623,157.265
C01338=1039.907,69.144,-88.261,169.648,38.624,157.265
C01339=1039.913,69.393,-88.280,169.650,38.624,157.266
C01340=1039.920,69.643,-88.298,169.652,38.625,157.266
C01341=1039.926,69.892,-88.317,169.655,38.626,157.266
C01342=1039.932,70.141,-88.334,169.656,38.626,157.266
C01343=1039.938,70.390,-88.353,169.658,38.627,157.266
C01344=1039.945,70.640,-88.370,169.660,38.628,157.266
C01345=1039.951,70.889,-88.389,169.662,38.628,157.267
C01346=1039.957,71.139,-88.407,169.664,38.629,157.267
C01347=1039.963,71.387,-88.425,169.666,38.629,157.267
C01348=1039.969,71.637,-88.443,169.667,38.630,157.267
C01349=1039.976,71.886,-88.462,169.669,38.630,157.267
C01350=1039.982,72.136,-88.480,169.672,38.631,157.267
C01351=1039.988,72.385,-88.498,169.674,38.632,157.268
C01352=1039.995,72.633,-88.515,169.676,38.632,157.268
C01353=1040.001,72.883,-88.534,169.678,38.633,157.268
C01354=1040.007,73.132,-88.552,169.679,38.634,157.268
C01355=1040.014,73.381,-88.570,169.681,38.634,157.268
C01356=1040.020,73.631,-88.588,169.683,38.635,157.268
C01357=1040.026,73.880,-88.607,169.686,38.635,157.268
C01358=1040.032,74.129,-88.625,169.688,38.636,157.269
C01359=1040.038,74.378,-88.643,169.690,38.636,157.269
C01360=1040.044,74.628,-88.662,169.692,38.637,157.269
C01361=1040.051,74.877,-88.680,169.693,38.638,157.269
C01362=1040.057,75.126,-88.698,169.695,38.638,157.269
C01363=1040.063,75.376,-88.717,169.697,38.639,157.269
C01364=1040.070,75.625,-88.734,169.700,38.639,157.270
C01365=1040.077,75.874,-88.753,169.702,38.640,157.270
C01366=1040.082,76.123,-88.771,169.704,38.640,157.270
C01367=1040.089,76.372,-88.789,169.705,38.641,157.270
C01368=1040.096,76.659,-88.811,169.708,38.642,157.270
C01369=1040.104,76.945,-88.832,169.710,38.643,157.271
C01370=1040.110,77.231,-88.853,169.712,38.643,157.271
C01371=1040.118,77.517,-88.874,169.715,38.644,157.271
C01372=1040.124,77.766,-88.892,169.717,38.644,157.271
C01373=1040.131,78.015,-88.911,169.719,38.645,157.271
C01374=1040.137,78.265,-88.929,169.720,38.646,157.271
C01375=1040.142,78.514,-88.948,169.722,38.647,157.272
C01376=1040.148,78.763,-88.966,169.724,38.647,157.272
C01377=1040.155,79.012,-88.985,169.726,38.648,157.272
C01378=1040.161,79.262,-89.003,169.729,38.648,157.272
C01379=1040.167,79.511,-89.022,169.731,38.649,157.272
C01380=1040.174,79.760,-89.040,169.732,38.650,157.272
C01381=1040.179,80.009,-89.059,169.734,38.650,157.273
C01382=1040.186,80.258,-89.078,169.736,38.651,157.273
C01383=1040.192,80.508,-89.096,169.738,38.651,157.273
C01384=1040.198,80.757,-89.115,169.741,38.653,157.273
C01385=1040.205,81.006,-89.133,169.742,38.653,157.273
C01386=1040.210,81.256,-89.153,169.744,38.654,157.273
C01387=1040.216,81.504,-89.171,169.746,38.654,157.274
C01388=1040.223,81.753,-89.189,169.748,38.655,157.274
C01389=1040.229,82.003,-89.207,169.750,38.656,157.274
C01390=1040.235,82.252,-89.226,169.752,38.656,157.274
C01391=1040.242,82.501,-89.245,169.754,38.657,157.274
C01392=1040.247,82.751,-89.264,169.756,38.658,157.274
C01393=1040.254,83.000,-89.283,169.758,38.658,157.275
C01394=1040.260,83.249,-89.301,169.760,38.659,157.275
C01395=1040.267,83.498,-89.320,169.762,38.660,157.275
C01396=1040.273,83.747,-89.339,169.764,38.660,157.275
C01397=1040.279,83.997,-89.358,169.765,38.661,157.275
C01398=1040.285,84.246,-89.376,169.768,38.661,157.275
C01399=1040.292,84.495,-89.395,169.770,38.662,157.276
C01400=1040.298,84.745,-89.413,169.772,38.663,157.276
C01401=1040.303,84.994,-89.432,169.774,38.664,157.276
C01402=1040.310,85.243,-89.451,169.776,38.664,157.276
C01403=1040.316,85.492,-89.470,169.777,38.665,157.276
C01404=1040.323,85.741,-89.488,169.779,38.665,157.276
C01405=1040.329,85.991,-89.507,169.782,38.666,157.277
C01406=1040.335,86.240,-89.526,169.784,38.666,157.277
C01407=1040.341,86.489,-89.545,169.786,38.667,157.277
C01408=1040.348,86.738,-89.563,169.788,38.668,157.277
C01409=1040.354,86.987,-89.582,169.790,38.668,157.277
C01410=1040.360,87.236,-89.601,169.791,38.669,157.277
C01411=1040.366,87.486,-89.620,169.793,38.670,157.278
C01412=1040.373,87.735,-89.639,169.796,38.670,157.278
C01413=1040.379,87.984,-89.657,169.798,38.671,157.278
C01414=1040.385,88.233,-89.676,169.800,38.672,157.278
C01415=1040.392,88.483,-89.696,169.802,38.672,157.278
C01416=1040.398,88.732,-89.715,169.803,38.673,157.278
C01417=1040.405,88.981,-89.734,169.805,38.673,157.279
C01418=1040.411,89.230,-89.752,169.807,38.674,157.279
C01419=1040.417,89.480,-89.771,169.810,38.674,157.279
C01420=1040.423,89.729,-89.790,169.812,38.675,157.279
C01421=1040.430,89.978,-89.809,169.814,38.676,157.279
C01422=1040.436,90.227,-89.827,169.816,38.677,157.280
C01423=1040.442,90.476,-89.847,169.817,38.677,157.280
C01424=1040.448,90.725,-89.865,169.819,38.678,157.280
C01425=1040.454,90.974,-89.885,169.822,38.679,157.280
C01426=1040.461,91.223,-89.904,169.824,38.679,157.280
C01427=1040.466,91.473,-89.923,169.826,38.680,157.280
C01428=1040.473,91.722,-89.942,169.828,38.680,157.281
C01429=1040.479,91.972,-89.961,169.829,38.682,157.281
C01430=1040.486,92.221,-89.981,169.831,38.682,157.281
C01431=1040.492,92.470,-90.000,169.833,38.683,157.281
C01432=1040.499,92.756,-90.022,169.836,38.684,157.281
C01433=1040.506,93.041,-90.044,169.838,38.684,157.282
C01434=1040.513,93.328,-90.065,169.840,38.685,157.282
C01435=1040.520,93.613,-90.088,169.842,38.686,157.282
C01436=1040.526,93.863,-90.107,169.844,38.686,157.282
C01437=1040.532,94.112,-90.126,169.846,38.687,157.282
C01438=1040.539,94.362,-90.145,169.849,38.688,157.283
C01439=1040.545,94.611,-90.165,169.851,38.689,157.283
C01440=1040.551,94.860,-90.184,169.853,38.689,157.283
C01441=1040.557,95.109,-90.203,169.855,38.690,157.283
C01442=1040.563,95.358,-90.222,169.856,38.691,157.283
C01443=1040.569,95.607,-90.242,169.858,38.691,157.283
C01444=1040.576,95.857,-90.260,169.860,38.692,157.284
C01445=1040.582,96.105,-90.280,169.863,38.692,157.284
C01446=1040.589,96.355,-90.299,169.865,38.694,157.284
C01447=1040.594,96.605,-90.318,169.867,38.694,157.284
C01448=1040.601,96.853,-90.338,169.868,38.695,157.284
C01449=1040.607,97.103,-90.357,169.870,38.695,157.284
C01450=1040.613,97.352,-90.376,169.872,38.696,157.285
C01451=1040.619,97.600,-90.396,169.875,38.697,157.285
C01452=1040.626,97.850,-90.415,169.877,38.697,157.285
C01453=1040.632,98.099,-90.435,169.879,38.698,157.285
C01454=1040.638,98.349,-90.454,169.881,38.698,157.285
C01455=1040.644,98.598,-90.472,169.882,38.700,157.286
C01456=1040.650,98.846,-90.492,169.884,38.700,157.286
C01457=1040.657,99.096,-90.511,169.886,38.701,157.286
C01458=1040.663,99.345,-90.531,169.889,38.701,157.286
C01459=1040.670,99.594,-90.550,169.891,38.702,157.286
C01460=1040.676,99.843,-90.570,169.893,38.703,157.286
C01461=1040.682,100.092,-90.589,169.895,38.703,157.287
C01462=1040.689,100.342,-90.609,169.896,38.704,157.287
C01463=1040.694,100.591,-90.628,169.898,38.705,157.287
C01464=1040.701,100.840,-90.648,169.901,38.706,157.287
C01465=1040.707,101.089,-90.667,169.903,38.706,157.287
C01466=1040.713,101.338,-90.687,169.905,38.707,157.287
C01467=1040.719,101.588,-90.706,169.907,38.708,157.288
C01468=1040.725,101.837,-90.726,169.909,38.708,157.288
C01469=1040.731,102.086,-90.745,169.910,38.709,157.288
C01470=1040.737,102.335,-90.765,169.913,38.710,157.288
C01471=1040.743,102.584,-90.785,169.915,38.711,157.288
C01472=1040.750,102.834,-90.805,169.917,38.711,157.289
C01473=1040.756,103.082,-90.824,169.919,38.712,157.289
C01474=1040.761,103.332,-90.844,169.921,38.713,157.289
C01475=1040.768,103.580,-90.863,169.922,38.713,157.289
C01476=1040.775,103.830,-90.883,169.925,38.715,157.289
C01477=1040.780,104.079,-90.903,169.927,38.715,157.290
C01478=1040.786,104.328,-90.923,169.929,38.716,157.290
C01479=1040.792,104.577,-90.943,169.931,38.717,157.290
C01480=1040.799,104.826,-90.961,169.933,38.717,157.290
C01481=1040.805,105.076,-90.982,169.935,38.718,157.290
C01482=1040.811,105.324,-91.002,169.937,38.719,157.291
C01483=1040.817,105.574,-91.021,169.939,38.719,157.291
C01484=1040.824,105.823,-91.041,169.941,38.720,157.291
C01485=1040.830,106.072,-91.061,169.943,38.721,157.291
C01486=1040.836,106.321,-91.080,169.945,38.722,157.291
C01487=1040.842,106.570,-91.100,169.947,38.722,157.292
C01488=1040.849,106.820,-91.120,169.949,38.723,157.292
C01489=1040.854,107.069,-91.139,169.951,38.724,157.292
C01490=1040.860,107.318,-91.159,169.953,38.724,157.292
C01491=1040.867,107.567,-91.180,169.955,38.725,157.292
C01492=1040.874,107.816,-91.199,169.957,38.726,157.293
C01493=1040.879,108.065,-91.218,169.959,38.727,157.293
C01494=1040.886,108.315,-91.238,169.961,38.727,157.293
C01495=1040.892,108.564,-91.258,169.964,38.728,157.293
C01496=1040.899,108.849,-91.281,169.966,38.729,157.293
C01497=1040.906,109.135,-91.304,169.968,38.729,157.293
C01498=1040.914,109.421,-91.326,169.970,38.730,157.294
C01499=1040.921,109.708,-91.349,169.972,38.731,157.294
C01500=1040.927,109.957,-91.369,169.975,38.732,157.294
C01501=1040.933,110.205,-91.389,169.977,38.733,157.294
C01502=1040.939,110.455,-91.410,169.979,38.733,157.294
C01503=1040.945,110.704,-91.429,169.981,38.734,157.295
C01504=1040.951,110.953,-91.449,169.983,38.735,157.295
C01505=1040.958,111.203,-91.469,169.985,38.735,157.295
C01506=1040.964,111.452,-91.489,169.988,38.736,157.295
C01507=1040.970,111.700,-91.509,169.989,38.737,157.295
C01508=1040.976,111.950,-91.529,169.991,38.738,157.296
C01509=1040.982,112.199,-91.549,169.993,38.739,157.296
C01510=1040.989,112.448,-91.570,169.995,38.739,157.296
C01511=1040.995,112.697,-91.590,169.997,38.740,157.296
C01512=1041.001,112.946,-91.610,170.000,38.741,157.296
C01513=1041.008,113.195,-91.630,170.002,38.741,157.297
C01514=1041.014,113.444,-91.650,170.004,38.742,157.297
C01515=1041.020,113.693,-91.670,170.005,38.743,157.297
C01516=1041.026,113.942,-91.690,170.007,38.744,157.297
C01517=1041.032,114.191,-91.710,170.009,38.745,157.297
C01518=1041.037,114.440,-91.731,170.012,38.745,157.298
C01519=1041.044,114.690,-91.751,170.014,38.746,157.298
C01520=1041.050,114.939,-91.771,170.016,38.747,157.298
C01521=1041.056,115.188,-91.791,170.018,38.748,157.298
C01522=1041.062,115.437,-91.812,170.019,38.749,157.298
C01523=1041.068,115.686,-91.832,170.022,38.750,157.299
C01524=1041.074,115.936,-91.852,170.024,38.750,157.299
C01525=1041.080,116.185,-91.872,170.026,38.751,157.299
C01526=1041.086,116.434,-91.893,170.028,38.752,157.299
C01527=1041.092,116.683,-91.913,170.030,38.753,157.300
C01528=1041.099,116.931,-91.934,170.032,38.754,157.300
C01529=1041.104,117.180,-91.954,170.034,38.755,157.300
C01530=1041.110,117.430,-91.974,170.036,38.755,157.300
C01531=1041.116,117.679,-91.994,170.038,38.756,157.300
C01532=1041.123,117.928,-92.015,170.040,38.757,157.301
C01533=1041.128,118.177,-92.035,170.042,38.758,157.301
C01534=1041.134,118.426,-92.055,170.045,38.759,157.301
C01535=1041.141,118.675,-92.076,170.047,38.760,157.301
C01536=1041.146,118.924,-92.097,170.049,38.760,157.301
C01537=1041.153,119.174,-92.117,170.051,38.761,157.302
C01538=1041.159,119.423,-92.137,170.052,38.762,157.302
C01539=1041.166,119.672,-92.157,170.054,38.762,157.302
C01540=1041.171,119.921,-92.179,170.057,38.764,157.302
C01541=1041.178,120.170,-92.199,170.059,38.764,157.302
C01542=1041.184,120.419,-92.219,170.061,38.765,157.303
C01543=1041.189,120.668,-92.240,170.063,38.766,157.303
C01544=1041.196,120.917,-92.261,170.065,38.767,157.303
C01545=1041.202,121.166,-92.281,170.068,38.767,157.303
C01546=1041.208,121.416,-92.301,170.070,38.769,157.304
C01547=1041.214,121.664,-92.321,170.071,38.769,157.304
C01548=1041.221,121.913,-92.342,170.073,38.770,157.304
C01549=1041.227,122.162,-92.362,170.075,38.771,157.304
C01550=1041.232,122.412,-92.383,170.077,38.771,157.304
C01551=1041.238,122.661,-92.403,170.080,38.772,157.305
C01552=1041.245,122.910,-92.424,170.082,38.773,157.305
C01553=1041.251,123.159,-92.445,170.084,38.774,157.305
C01554=1041.257,123.408,-92.465,170.086,38.775,157.305
C01555=1041.264,123.656,-92.486,170.088,38.776,157.305
C01556=1041.269,123.906,-92.507,170.091,38.776,157.306
C01557=1041.275,124.155,-92.527,170.093,38.777,157.306
C01558=1041.282,124.404,-92.548,170.095,38.778,157.306
C01559=1041.288,124.654,-92.569,170.096,38.779,157.306
C01560=1041.295,124.939,-92.592,170.099,38.780,157.306
C01561=1041.302,125.225,-92.616,170.102,38.781,157.307
C01562=1041.309,125.511,-92.639,170.104,38.781,157.307
C01563=1041.316,125.797,-92.663,170.106,38.782,157.307
C01564=1041.323,126.046,-92.684,170.108,38.783,157.307
C01565=1041.329,126.295,-92.705,170.110,38.784,157.308
C01566=1041.335,126.544,-92.725,170.112,38.785,157.308
C01567=1041.341,126.792,-92.746,170.115,38.786,157.308
C01568=1041.351,127.151,-92.775,170.118,38.787,157.308
C01569=1041.359,127.509,-92.806,170.121,38.788,157.309
C01570=1041.368,127.867,-92.835,170.124,38.789,157.309
C01571=1041.377,128.225,-92.865,170.127,38.790,157.309
C01572=1041.383,128.474,-92.885,170.129,38.791,157.309
C01573=1041.390,128.723,-92.906,170.131,38.792,157.310
C01574=1041.396,128.972,-92.927,170.133,38.792,157.310
C01575=1041.402,129.221,-92.948,170.135,38.793,157.310
C01576=1041.408,129.470,-92.969,170.138,38.794,157.310
C01577=1041.415,129.719,-92.990,170.140,38.794,157.310
C01578=1041.421,129.968,-93.010,170.142,38.795,157.311
C01579=1041.427,130.217,-93.032,170.144,38.796,157.311
C01580=1041.434,130.467,-93.052,170.146,38.797,157.311
C01581=1041.440,130.715,-93.073,170.149,38.798,157.311
C01582=1041.446,130.965,-93.094,170.151,38.798,157.311
C01583=1041.453,131.214,-93.115,170.153,38.799,157.312
C01584=1041.459,131.462,-93.136,170.155,38.800,157.312
C01585=1041.465,131.712,-93.156,170.157,38.801,157.312
C01586=1041.471,131.960,-93.177,170.160,38.802,157.312
C01587=1041.477,132.210,-93.199,170.162,38.803,157.313
C01588=1041.484,132.459,-93.219,170.164,38.804,157.313
C01589=1041.489,132.708,-93.241,170.166,38.804,157.313
C01590=1041.495,132.957,-93.262,170.168,38.805,157.313
C01591=1041.502,133.206,-93.283,170.169,38.806,157.313
C01592=1041.507,133.455,-93.304,170.172,38.807,157.314
C01593=1041.514,133.704,-93.326,170.174,38.808,157.314
C01594=1041.520,133.953,-93.346,170.176,38.809,157.314
C01595=1041.526,134.202,-93.367,170.178,38.810,157.314
C01596=1041.532,134.451,-93.389,170.180,38.810,157.315
C01597=1041.539,134.700,-93.410,170.183,38.811,157.315
C01598=1041.544,134.949,-93.430,170.185,38.812,157.315
C01599=1041.550,135.198,-93.452,170.187,38.813,157.315
C01600=1041.557,135.447,-93.473,170.189,38.814,157.315
C01601=1041.563,135.696,-93.494,170.191,38.815,157.316
C01602=1041.569,135.945,-93.516,170.194,38.816,157.316
C01603=1041.575,136.195,-93.537,170.196,38.816,157.316
C01604=1041.581,136.443,-93.558,170.198,38.818,157.316
C01605=1041.587,136.692,-93.579,170.200,38.818,157.317
C01606=1041.593,136.941,-93.601,170.202,38.819,157.317
C01607=1041.600,137.190,-93.622,170.205,38.820,157.317
C01608=1041.606,137.439,-93.643,170.207,38.821,157.317
C01609=1041.612,137.689,-93.664,170.209,38.822,157.318
C01610=1041.618,137.938,-93.686,170.211,38.822,157.318
C01611=1041.625,138.187,-93.707,170.213,38.824,157.318
C01612=1041.630,138.435,-93.728,170.216,38.824,157.318
C01613=1041.636,138.684,-93.750,170.218,38.825,157.318
C01614=1041.643,138.934,-93.771,170.220,38.826,157.319
C01615=1041.649,139.182,-93.792,170.222,38.827,157.319
C01616=1041.655,139.431,-93.814,170.224,38.828,157.319
C01617=1041.661,139.680,-93.835,170.227,38.829,157.319
C01618=1041.667,139.929,-93.857,170.229,38.830,157.320
C01619=1041.673,140.178,-93.878,170.231,38.831,157.320
C01620=1041.679,140.391,-93.896,170.232,38.831,157.320
C01621=1041.683,140.604,-93.915,170.234,38.832,157.320
C01622=1041.689,140.818,-93.933,170.237,38.833,157.320
C01623=1041.694,141.030,-93.951,170.239,38.833,157.321
C01624=1041.699,141.243,-93.969,170.240,38.835,157.321
C01625=1041.704,141.456,-93.989,170.242,38.835,157.321
C01626=1041.710,141.669,-94.007,170.244,38.836,157.321
C01627=1041.715,141.881,-94.025,170.245,38.837,157.321
C01628=1041.721,142.130,-94.046,170.248,38.838,157.322
C01629=1041.727,142.380,-94.068,170.250,38.839,157.322
C01630=1041.733,142.629,-94.090,170.252,38.840,157.322
C01631=1041.739,142.878,-94.111,170.254,38.841,157.322
C01632=1041.745,143.126,-94.132,170.256,38.841,157.323
C01633=1041.751,143.376,-94.154,170.259,38.842,157.323
C01634=1041.758,143.624,-94.176,170.261,38.844,157.323
C01635=1041.764,143.873,-94.198,170.263,38.844,157.323
C01636=1041.770,144.123,-94.220,170.265,38.845,157.324
C01637=1041.775,144.371,-94.241,170.268,38.846,157.324
C01638=1041.782,144.620,-94.263,170.270,38.847,157.324
C01639=1041.788,144.870,-94.284,170.272,38.848,157.324
C01640=1041.794,145.119,-94.306,170.274,38.849,157.325
C01641=1041.800,145.367,-94.328,170.276,38.850,157.325
C01642=1041.807,145.617,-94.350,170.279,38.851,157.325
C01643=1041.813,145.865,-94.371,170.282,38.852,157.325
C01644=1041.819,146.114,-94.392,170.284,38.852,157.325
C01645=1041.825,146.363,-94.414,170.286,38.853,157.326
C01646=1041.831,146.612,-94.435,170.289,38.855,157.326
C01647=1041.838,146.861,-94.458,170.291,38.855,157.326
C01648=1041.844,147.110,-94.479,170.293,38.856,157.326
C01649=1041.850,147.359,-94.501,170.295,38.857,157.327
C01650=1041.856,147.609,-94.523,170.297,38.858,157.327
C01651=1041.861,147.857,-94.545,170.300,38.859,157.327
C01652=1041.868,148.106,-94.567,170.302,38.860,157.327
C01653=1041.874,148.355,-94.589,170.304,38.861,157.328
C01654=1041.880,148.604,-94.611,170.306,38.862,157.328
C01655=1041.886,148.853,-94.633,170.308,38.863,157.328
C01656=1041.893,149.102,-94.654,170.311,38.864,157.328
C01657=1041.899,149.351,-94.677,170.313,38.865,157.329
C01658=1041.905,149.600,-94.699,170.315,38.866,157.329
C01659=1041.910,149.849,-94.720,170.317,38.867,157.329
C01660=1041.917,150.097,-94.742,170.320,38.868,157.329
C01661=1041.923,150.347,-94.764,170.322,38.869,157.330
C01662=1041.929,150.596,-94.786,170.324,38.870,157.330
C01663=1041.935,150.845,-94.809,170.326,38.871,157.330
C01664=1041.941,151.094,-94.830,170.328,38.872,157.330
C01665=1041.947,151.342,-94.853,170.331,38.873,157.331
C01666=1041.953,151.592,-94.874,170.333,38.874,157.331
C01667=1041.960,151.841,-94.896,170.335,38.875,157.331
C01668=1041.965,152.090,-94.919,170.338,38.876,157.332
C01669=1041.971,152.339,-94.940,170.341,38.877,157.332
C01670=1041.978,152.588,-94.963,170.343,38.878,157.332
C01671=1041.984,152.837,-94.984,170.345,38.879,157.332
C01672=1041.990,153.085,-95.006,170.347,38.880,157.333
C01673=1041.995,153.334,-95.029,170.350,38.881,157.333
C01674=1042.002,153.583,-95.051,170.352,38.882,157.333
C01675=1042.008,153.832,-95.073,170.354,38.883,157.333
C01676=1042.014,154.081,-95.095,170.356,38.884,157.334
C01677=1042.020,154.330,-95.117,170.358,38.884,157.334
C01678=1042.026,154.579,-95.140,170.361,38.886,157.334
C01679=1042.033,154.828,-95.161,170.363,38.887,157.334
C01680=1042.038,155.077,-95.184,170.365,38.888,157.335
C01681=1042.045,155.325,-95.207,170.367,38.889,157.335
C01682=1042.051,155.575,-95.228,170.370,38.890,157.335
C01683=1042.057,155.823,-95.251,170.373,38.891,157.336
C01684=1042.063,156.073,-95.273,170.375,38.892,157.336
C01685=1042.069,156.321,-95.295,170.377,38.893,157.336
C01686=1042.075,156.570,-95.318,170.380,38.894,157.336
C01687=1042.081,156.819,-95.340,170.382,38.895,157.337
C01688=1042.089,157.105,-95.366,170.384,38.896,157.337
C01689=1042.095,157.390,-95.391,170.387,38.897,157.337
C01690=1042.102,157.675,-95.417,170.390,38.898,157.337
C01691=1042.109,157.961,-95.443,170.393,38.899,157.338
C01692=1042.116,158.209,-95.465,170.395,38.900,157.338
C01693=1042.122,158.459,-95.487,170.397,38.902,157.338
C01694=1042.127,158.708,-95.510,170.400,38.903,157.339
C01695=1042.134,158.956,-95.532,170.402,38.904,157.339
C01696=1042.140,159.205,-95.555,170.404,38.905,157.339
C01697=1042.146,159.454,-95.577,170.406,38.906,157.339
C01698=1042.152,159.703,-95.599,170.409,38.907,157.340
C01699=1042.158,159.952,-95.622,170.411,38.908,157.340
C01700=1042.165,160.200,-95.644,170.414,38.909,157.340
C01701=1042.170,160.450,-95.666,170.416,38.910,157.340
C01702=1042.176,160.699,-95.689,170.419,38.911,157.341
C01703=1042.182,160.947,-95.712,170.421,38.912,157.341
C01704=1042.188,161.196,-95.735,170.423,38.913,157.341
C01705=1042.194,161.445,-95.758,170.425,38.915,157.342
C01706=1042.199,161.694,-95.781,170.428,38.916,157.342
C01707=1042.205,161.943,-95.803,170.430,38.917,157.342
C01708=1042.212,162.191,-95.826,170.432,38.918,157.343
C01709=1042.217,162.440,-95.849,170.434,38.919,157.343
C01710=1042.223,162.691,-95.871,170.437,38.921,157.343
C01711=1042.229,162.940,-95.894,170.439,38.922,157.343
C01712=1042.235,163.188,-95.917,170.442,38.923,157.344
C01713=1042.241,163.437,-95.940,170.444,38.924,157.344
C01714=1042.247,163.686,-95.963,170.447,38.925,157.344
C01715=1042.253,163.935,-95.985,170.449,38.926,157.345
C01716=1042.258,164.184,-96.008,170.451,38.927,157.345
C01717=1042.265,164.432,-96.031,170.454,38.929,157.345
C01718=1042.271,164.681,-96.054,170.456,38.930,157.346
C01719=1042.276,164.930,-96.077,170.458,38.931,157.346
C01720=1042.282,165.179,-96.100,170.460,38.932,157.346
C01721=1042.288,165.428,-96.123,170.464,38.933,157.346
C01722=1042.295,165.676,-96.146,170.466,38.935,157.347
C01723=1042.300,165.925,-96.169,170.468,38.936,157.347
C01724=1042.307,166.174,-96.192,170.470,38.937,157.347
C01725=1042.312,166.423,-96.215,170.473,38.938,157.348
C01726=1042.318,166.672,-96.238,170.475,38.939,157.348
C01727=1042.325,166.921,-96.260,170.477,38.940,157.348
C01728=1042.330,167.170,-96.283,170.481,38.942,157.349
C01729=1042.336,167.418,-96.306,170.483,38.943,157.349
C01730=1042.342,167.667,-96.329,170.485,38.944,157.349
C01731=1042.348,167.917,-96.352,170.487,38.945,157.349
C01732=1042.354,168.165,-96.376,170.490,38.946,157.350
C01733=1042.361,168.414,-96.398,170.492,38.947,157.350
C01734=1042.366,168.663,-96.421,170.494,38.949,157.350
C01735=1042.372,168.912,-96.444,170.497,38.950,157.351
C01736=1042.378,169.161,-96.467,170.500,38.951,157.351
C01737=1042.384,169.410,-96.490,170.502,38.952,157.351
C01738=1042.390,169.658,-96.514,170.504,38.954,157.352
C01739=1042.397,169.907,-96.536,170.506,38.955,157.352
C01740=1042.402,170.156,-96.559,170.509,38.956,157.352
C01741=1042.408,170.405,-96.582,170.512,38.957,157.352
C01742=1042.415,170.654,-96.606,170.514,38.958,157.353
C01743=1042.420,170.903,-96.629,170.517,38.959,157.353
C01744=1042.426,171.152,-96.652,170.519,38.960,157.353
C01745=1042.433,171.400,-96.675,170.521,38.961,157.354
C01746=1042.439,171.649,-96.699,170.524,38.962,157.354
C01747=1042.445,171.898,-96.722,170.527,38.964,157.354
C01748=1042.451,172.147,-96.745,170.529,38.965,157.355
C01749=1042.457,172.396,-96.767,170.531,38.966,157.355
C01750=1042.463,172.645,-96.792,170.533,38.967,157.355
C01751=1042.469,172.894,-96.814,170.537,38.968,157.355
C01752=1042.477,173.178,-96.841,170.539,38.970,157.356
C01753=1042.483,173.463,-96.867,170.542,38.971,157.356
C01754=1042.490,173.748,-96.894,170.545,38.972,157.356
C01755=1042.497,174.033,-96.921,170.548,38.974,157.357
C01756=1042.503,174.282,-96.944,170.550,38.975,157.357
C01757=1042.509,174.530,-96.968,170.553,38.976,157.357
C01758=1042.515,174.780,-96.991,170.555,38.977,157.358
C01759=1042.522,175.028,-97.013,170.558,38.978,157.358
C01760=1042.528,175.277,-97.037,170.560,38.980,157.358
C01761=1042.534,175.526,-97.060,170.563,38.981,157.359
C01762=1042.540,175.774,-97.084,170.565,38.982,157.359
C01763=1042.546,176.023,-97.107,170.568,38.983,157.359
C01764=1042.553,176.272,-97.131,170.570,38.985,157.360
C01765=1042.558,176.521,-97.154,170.573,38.986,157.360
C01766=1042.564,176.770,-97.177,170.575,38.987,157.360
C01767=1042.572,177.019,-97.200,170.578,38.988,157.360
C01768=1042.577,177.268,-97.223,170.581,38.990,157.361
C01769=1042.584,177.517,-97.247,170.583,38.991,157.361
C01770=1042.590,177.765,-97.271,170.585,38.992,157.361
C01771=1042.596,178.014,-97.294,170.588,38.993,157.362
C01772=1042.602,178.263,-97.318,170.591,38.994,157.362
C01773=1042.608,178.512,-97.341,170.593,38.995,157.362
C01774=1042.615,178.761,-97.365,170.596,38.997,157.363
C01775=1042.620,179.010,-97.388,170.599,38.998,157.363
C01776=1042.626,179.258,-97.411,170.601,38.999,157.363
C01777=1042.634,179.507,-97.434,170.603,39.000,157.364
C01778=1042.640,179.755,-97.458,170.606,39.001,157.364
C01779=1042.646,180.004,-97.482,170.609,39.002,157.364
C01780=1042.652,180.253,-97.505,170.611,39.004,157.365
C01781=1042.659,180.502,-97.529,170.614,39.005,157.365
C01782=1042.664,180.751,-97.552,170.617,39.006,157.365
C01783=1042.671,181.000,-97.576,170.619,39.007,157.365
C01784=1042.677,181.248,-97.599,170.621,39.008,157.366
C01785=1042.683,181.498,-97.623,170.624,39.009,157.366
C01786=1042.689,181.746,-97.646,170.627,39.011,157.366
C01787=1042.696,181.995,-97.670,170.629,39.012,157.367
C01788=1042.702,182.244,-97.693,170.632,39.013,157.367
C01789=1042.708,182.493,-97.717,170.634,39.014,157.367
C01790=1042.715,182.741,-97.740,170.637,39.015,157.368
C01791=1042.721,182.991,-97.764,170.640,39.017,157.368
C01792=1042.727,183.239,-97.787,170.642,39.018,157.368
C01793=1042.734,183.488,-97.811,170.645,39.019,157.369
C01794=1042.740,183.736,-97.835,170.648,39.020,157.369
C01795=1042.746,183.986,-97.860,170.650,39.022,157.369
C01796=1042.752,184.234,-97.883,170.653,39.023,157.370
C01797=1042.758,184.484,-97.907,170.656,39.025,157.370
C01798=1042.764,184.732,-97.931,170.658,39.026,157.370
C01799=1042.769,184.981,-97.955,170.661,39.028,157.371
C01800=1042.776,185.230,-97.979,170.663,39.029,157.371
C01801=1042.781,185.478,-98.003,170.666,39.030,157.371
C01802=1042.788,185.727,-98.027,170.669,39.032,157.372
C01803=1042.793,185.976,-98.052,170.671,39.033,157.372
C01804=1042.800,186.225,-98.076,170.674,39.034,157.372
C01805=1042.805,186.473,-98.100,170.677,39.036,157.373
C01806=1042.811,186.722,-98.124,170.679,39.037,157.373
C01807=1042.817,186.971,-98.148,170.681,39.039,157.374
C01808=1042.823,187.220,-98.172,170.684,39.040,157.374
C01809=1042.829,187.468,-98.197,170.687,39.042,157.374
C01810=1042.835,187.717,-98.221,170.689,39.043,157.375
C01811=1042.841,187.966,-98.245,170.693,39.044,157.375
C01812=1042.847,188.215,-98.269,170.695,39.046,157.375
